           IF #rdrec.valid = TRUE THEN
               // store information of data record
               #readdata[0] := DINT_TO_BYTE(#RDREC_Function.INDEX); // ID of data record
               #readdata[1] := UINT_TO_BYTE(#rdrec.len);    // Length of data record
               #idpos := DINT#8;   // set start position within data
               MOVE_BLK(IN := #recorddata[0],
                        COUNT := #rdrec.len,
                        OUT => #readdata[#idpos]);
               #readlength := UINT_TO_INT(#rdrec.len);
               #sequencecontrol := 11;

           ELSIF #rdrec.error = TRUE THEN
               #ERROR := TRUE;
               #SF_STATUS := #rdrec.status;
               #sequencecontrol := 99; // function aborted with error
           ELSE
               ;
           END_IF; // store information of data record

       11:  // evaluate Consistency Check = Index 230d    
           #RDREC_Function(REQ := FALSE,
                           ID := #ID,
                           INDEX := DINT#230,
                           MLEN := UINT#0,
                           VALID => #rdrec.valid,
                           BUSY => #rdrec.busy,
                           ERROR => #rdrec.error,
                           STATUS => #rdrec.status,
                           LEN => #rdrec.len,
                           RECORD := #recorddata);

           IF #rdrec.valid = FALSE THEN
               #sequencecontrol := 12;
           ELSE
               ;
           END_IF;

       12:  // read Expected Port Configuration = Index 220d
           #STATUS := DW#16#00010220;
           #RDREC_Function(REQ := TRUE,
                           ID := #ID,
                           INDEX := DINT#220,
                           MLEN := UINT#0,
                           VALID => #rdrec.valid,
                           BUSY => #rdrec.busy,
                           ERROR => #rdrec.error,
                           STATUS => #rdrec.status,
                           LEN => #rdrec.len,
                           RECORD := #recorddata);

           IF #rdrec.valid = TRUE THEN
               // store information of data record
               #readdata[2] := DINT_TO_BYTE(#RDREC_Function.INDEX); // ID of data record
               #readdata[3] := UINT_TO_BYTE(#rdrec.len);    // Length of data record
               #idpos := #idpos + BYTE_TO_DINT(#readdata[1]);   // set start position within data
               MOVE_BLK(IN := #recorddata[0],
                        COUNT := #rdrec.len,
                        OUT => #readdata[#idpos]);
               #readlength := #readlength + UINT_TO_INT(#rdrec.len);
               #sequencecontrol := 13;

           ELSIF #rdrec.error = TRUE THEN
               #ERROR := TRUE;
               #SF_STATUS := #rdrec.status;
               #sequencecontrol := 99; // function aborted with error
           ELSE
               ;
           END_IF;

       13:  // evaluate Expected Port Configuration = Index 220d    
           #RDREC_Function(REQ := FALSE,
                           ID := #ID,
                           INDEX := DINT#220,
                           MLEN := UINT#0,
                           VALID => #rdrec.valid,
                           BUSY => #rdrec.busy,
                           ERROR => #rdrec.error,
                           STATUS => #rdrec.status,
                           LEN => #rdrec.len,
                           RECORD := #recorddata);
           IF #rdrec.valid = FALSE THEN
               #sequencecontrol := 14;
           END_IF;

       14:  // read IO Mapping = Index 222d
           #STATUS := DW#16#00010222;
           #RDREC_Function(REQ := TRUE,
                           ID := #ID,
                           INDEX := DINT#222,
                           MLEN := UINT#0,
                           VALID => #rdrec.valid,
                           BUSY => #rdrec.busy,
                           ERROR => #rdrec.error,
                           STATUS => #rdrec.status,
                           LEN => #rdrec.len,
                           RECORD := #recorddata);

           IF #rdrec.valid = TRUE THEN
               // store information of data record
               #readdata[4] := DINT_TO_BYTE(#RDREC_Function.INDEX); // ID of data record
               #readdata[5] := UINT_TO_BYTE(#rdrec.len);    // Length of data record
               #idpos := #idpos + BYTE_TO_DINT(#readdata[3]);   // set start position within data
               MOVE_BLK(IN := #recorddata[0],
                        COUNT := #rdrec.len,
                        OUT => #readdata[#idpos]);
               #readlength := #readlength + UINT_TO_INT(#rdrec.len);
               #sequencecontrol := 15;

           ELSIF #rdrec.error = TRUE THEN
               #ERROR := TRUE;
               #SF_STATUS := #rdrec.status;
               #sequencecontrol := 99; // function aborted with error
           ELSE
               ;
           END_IF;

       15:  // evaluate IO Mapping = Index 222d    
           #RDREC_Function(REQ := FALSE,
                           ID := #ID,
                           INDEX := DINT#222,
                           MLEN := UINT#0,
                           VALID => #rdrec.valid,
                           BUSY => #rdrec.busy,
                           ERROR => #rdrec.error,
                           STATUS => #rdrec.status,
                           LEN => #rdrec.len,
                           RECORD := #recorddata);
           IF #rdrec.valid = FALSE THEN
               #sequencecontrol := 16;
           END_IF;

       16:  // BACKUP complete and valid
           #RECORD_DATA := #readdata;
           #DONE_VALID := TRUE;
           #BUSY := FALSE;
           #ERROR := FALSE;
           #STATUS := DW#16#00010000;
           #SF_STATUS := DW#16#00000000;
           #RD_LEN := #readlength + INT#8;

           #sequencecontrol := 98;

   (*---------------------------------------------------------------------------------------------------------------------
               Write master parameter = RESTORE
   ---------------------------------------------------------------------------------------------------------------------*)
       20: // write Expected Port Configuration = Index 220d
           #STATUS := DW#16#00020220;
           #idpos := DINT#8 + BYTE_TO_DINT(#writedata[1]);  // position of data record 
           #wrrec.len := BYTE_TO_UINT(#writedata[3]);   // length of data record
           MOVE_BLK(IN := #writedata[#idpos],
                    COUNT := #wrrec.len,
                    OUT => #recorddata[0]);
           #WRREC_Function(REQ := TRUE,
                           ID := #ID,
                           INDEX := BYTE_TO_DINT(#writedata[2]),
                           LEN := #wrrec.len,
                           DONE => #wrrec.done,
                           BUSY => #wrrec.busy,
                           ERROR => #wrrec.error,
                           STATUS => #wrrec.status,
                           RECORD := #recorddata);
           // wait for finish writing Expected Port Configuration = Index 220d                
           IF #wrrec.done = TRUE THEN
               #sequencecontrol := 21;
           ELSIF #wrrec.error = TRUE THEN
               #ERROR := TRUE;
               #SF_STATUS := #wrrec.status;
               #sequencecontrol := 99; // function aborted with error
           ELSE
               ;
           END_IF;

       21:  // writing Expected Port Configuration finished    
           #WRREC_Function(REQ := FALSE,
                           ID := #ID,
                           INDEX := BYTE_TO_DINT(#writedata[2]),
                           LEN := #wrrec.len,
                           DONE => #wrrec.done,
                           BUSY => #wrrec.busy,
                           ERROR => #wrrec.error,
                           STATUS => #wrrec.status,
                           RECORD := #recorddata);
           IF #wrrec.done = FALSE THEN
               #sequencecontrol := 22;
           END_IF;

       22:  // write IO Mapping = Index 222d
           #STATUS := DW#16#00020222;
           #idpos := DINT#8 + BYTE_TO_DINT(#writedata[1]) + BYTE_TO_DINT(#writedata[3]);  // position of data record 
           #wrrec.len := BYTE_TO_UINT(#writedata[5]);   // length of data record
           MOVE_BLK(IN := #writedata[#idpos],
                    COUNT := #wrrec.len,
                    OUT => #recorddata[0]);
           #WRREC_Function(REQ := TRUE,
                           ID := #ID,
                           INDEX := BYTE_TO_DINT(#writedata[4]),
                           LEN := #wrrec.len,
                           DONE => #wrrec.done,
                           BUSY => #wrrec.busy,
                           ERROR => #wrrec.error,
                           STATUS => #wrrec.status,
                           RECORD := #recorddata);
           // wait for finish writing IO Mapping = Index 222d                
           IF #wrrec.done = TRUE THEN
               #sequencecontrol := 23;
           ELSIF #wrrec.error = TRUE THEN
               #ERROR := TRUE;
               #SF_STATUS := #wrrec.status;
               #sequencecontrol := 99;
           ELSE
               ;
           END_IF;

       23:  // writing IO Mapping finished    
           #WRREC_Function(REQ := FALSE,
                           ID := #ID,
                           INDEX := BYTE_TO_DINT(#writedata[4]),
                           LEN := #wrrec.len,
                           DONE => #wrrec.done,
                           BUSY => #wrrec.busy,
                           ERROR => #wrrec.error,
                           STATUS => #wrrec.status,
                           RECORD := #recorddata);
           IF #wrrec.done = FALSE THEN
               #sequencecontrol := 24;
           END_IF;

       24:  // write Consistency Check = Index 230d
           #STATUS := DW#16#00020230;
           #idpos := DINT#8;  // position of data record 
           #wrrec.len := BYTE_TO_UINT(#writedata[1]);   // length of data record
           MOVE_BLK(IN := #writedata[#idpos],
                    COUNT := #wrrec.len,
                    OUT => #recorddata[0]);
           #WRREC_Function(REQ := TRUE,
                           ID := #ID,
                           INDEX := BYTE_TO_DINT(#writedata[0]),
                           LEN := #wrrec.len,
                           DONE => #wrrec.done,
                           BUSY => #wrrec.busy,
                           ERROR => #wrrec.error,
                           STATUS => #wrrec.status,
                           RECORD := #recorddata);
           // wait for finish writing Consistency Check = Index 230d               
           IF #wrrec.done = TRUE THEN
               #sequencecontrol := 25;
           ELSIF #wrrec.error = TRUE THEN
               #ERROR := TRUE;
               #SF_STATUS := #wrrec.status;
               #sequencecontrol := 99;
           ELSE
               ;
           END_IF;

       25:  // writing ConsistencyCheck finished    
           #WRREC_Function(REQ := FALSE,
                           ID := #ID,
                           INDEX := BYTE_TO_DINT(#writedata[0]),
                           LEN := #wrrec.len,
                           DONE => #wrrec.done,
                           BUSY => #wrrec.busy,
                           ERROR => #wrrec.error,
                           STATUS => #wrrec.status,
                           RECORD := #recorddata);
           IF #wrrec.done = FALSE THEN
               #sequencecontrol := 26;
           END_IF;

       26:  // RESTORE complete and valid
           #DONE_VALID := TRUE;
           #BUSY := FALSE;
           #ERROR := FALSE;
           #STATUS := DW#16#00020000;
           #SF_STATUS := DW#16#00000000;
           #RD_LEN := INT#0;

           #sequencecontrol := 98;

   (*---------------------------------------------------------------------------------------------------------------------
               END of SEQUENCE CONTROL
   ---------------------------------------------------------------------------------------------------------------------*)
       98: // Function complete and finish without error
           #RDREC_Function(REQ := FALSE,
                           RECORD := #recorddata);
           #WRREC_Function(REQ := FALSE);
           IF #REQ = FALSE THEN
               #DONE_VALID := FALSE;
               #STATUS := DW#16#00000000;
               #SF_STATUS := DW#16#00000000;
               #RD_LEN := INT#0;
               #sequencecontrol := 0;
               #typeofrequest := 0;
           END_IF;

       99: // Function aborted with error
           #RDREC_Function(REQ := FALSE,
                           RECORD := #recorddata);
           #WRREC_Function(REQ := FALSE);
           #DONE_VALID := FALSE;
           #BUSY := FALSE;
           #RD_LEN := INT#0;
           #sequencecontrol := 0;
           #typeofrequest := 0;

       ELSE  // no relevant case, ready for new request
           ;
   END_CASE;
END_FUNCTION_BLOCK

FUNCTION_BLOCK "IO_LINK_DEVICE"   // FB50001, SCL
{ S7_Optimized_Access := 'TRUE' }
AUTHOR : SUP_FA
FAMILY : IO-Link
VERSION : 3.0
   VAR_INPUT
      REQ : Bool;   // Request Function / Neuer Auftrag
      ID : Hw_Io;   // Hardwarekennung des IOL-Master Moduls (HW_IO) aus HW-Konfiguration
      CAP : DInt := DINT#0;   // Client Access Point (CAP), bei ET200 immer 227 dez
      RD_WR : Bool;   // Lese und Schreibzugriff auf IO-Link Device 0: Lesen, 1: schreiben
      PORT : Int := INT#0;   // Port/ Kanalnummer an dem das IO-Link Device betrieben wird. (ET200 = 1 .. 4)
      IOL_INDEX : Int := INT#0;   // Adressparameter Index (IO-Link Device) 0..32767 IOL-D, 65535 port functions
      IOL_SUBINDEX : Int := INT#0;   // Adressparameter Subindex (IO-Link Device) 0 ges. Record; 1-255 einz. Parameter
      LEN : Int := INT#0;   // Länge der zu schreibenden Daten (Nettodaten)
   END_VAR
   VAR_OUTPUT
      DONE_VALID : Bool;   // Gültigkeit 0: Daten nicht gültig; 1: Daten gültig
      BUSY : Bool;   // 0: Auftrag abgeschlossen 1: Auftrag in Bearbeitung
      ERROR : Bool;   // Fehler Flag 0: kein Fehler; 1: Abbruch der Funktion mit Fehler
      STATUS : DWord := DW#16#00000000;   // DP/ PNIO - Fehlerstatus; ERROR Flag = 1 - detaillierter Kommunikationsfehlerstatus
      IOL_STATUS : DWord := DW#16#00000000;   // IO-Link Fehlerstatus; ERROR Flag = 1 - detaillierte IO-Link Fehlerstatus
      RD_LEN : Int := INT#0;   // Länge des gelesenen Datensatzes (Anzahl Bytes)
   END_VAR
   VAR_IN_OUT
      RECORD_IOL_DATA : Array[0..231] of Byte;   // Datenbereich für LESEN / SCHREIBEN (max. 232 Byte)
   END_VAR
   VAR
      RDREC_Function : RDREC;   // Funktion Datensatz lesen (ehemals SFB52)
      WRREC_Function : WRREC;   // Funktion Datensatz schreiben (ehemals SFB53)
      TP_poll : TP_TIME;   // Pollzeit für "Datensatz lesen"
      TON_monitoring : TON_TIME;   // Überwachungszeit für Aufträge
      rdrec : Struct   // interne Struktur für RDREC
         valid : Bool;
         busy : Bool;
         error : Bool;
         status : DWord;
         length : UInt;
      END_STRUCT;
      wrrec : Struct   // interne Struktur für WRREC
         length : UInt;
         done : Bool;
         busy : Bool;
         error : Bool;
         status : DWord;
      END_STRUCT;
      read : Struct   // Datenbereich für Lesedaten
         header : Struct
            CALL : Struct
               Extended_Function_Num : Byte := 16#8;
               Port : Byte;
               FI_Index : Word := 16#FE4A;
            END_STRUCT;
            IOL : Struct
               Control : Byte;
               Index_HighByte : Byte;
               Index_LowByte : Byte;
               Subindex : Byte;
            END_STRUCT;
         END_STRUCT;
         data : Array[0..231] of Byte;
      END_STRUCT;
      write : Struct   // Datenbereich für Schreibdaten
         header : Struct
            CALL : Struct
               Extended_Function_Num : Byte := 16#8;
               Port : Byte;
               FI_Index : Word := 16#FE4A;
            END_STRUCT;
            IOL : Struct
               Control : Byte;
               Index_HighByte : Byte;
               Index_LowByte : Byte;
               Subindex : Byte;
            END_STRUCT;
         END_STRUCT;
         data : Array[0..231] of Byte;
      END_STRUCT;
      sequencecontrol : Int := INT#0;
      typeofrequest : Int := INT#0;
      R_TRIG_REQ : Bool;   // Impuls für neuen Auftrag starten
      R_TRIG_REQ_old : Bool;   // Flankenmerker
      F_TRIG_poll : Bool;   // Impuls für Pollen "Datensatz lesen"
      F_TRIG_poll_old : Bool;   // Flankenmerker
   END_VAR
   VAR_TEMP
      retval : Int;   // Variable für Rückgabewerte von Funktionen
      tmpWORD : Word;   // Datentyp WORD zur temporären Verwendung
      tmpDWORD : DWord;   // Datentyp DWORD zur temporären Verwendung
      tmpINT : Int;   // Datentyp INT zur temporären Verwendung
      i : Int;   // Laufvariable für for-Schleifen
   END_VAR
BEGIN
   (*---------------------------------------------------------------------------------------------------------------------
   SIEMENS AG
   ©Copyright 2015. All Rights Reserved.
   -----------------------------------------------------------------------------------------------------------------------
   Limitation of liability
   This software was developed with largest care. However, the author can not guarantee, that the software runs under
   each version of STEP7 on each PLC flawlessly.
   There is no warranty for the software, to the extent permitted by applicable law. The copyright holder provides the
   software "as is" without warranty of any kind, either expressed or implied, including, but not limited to, the implied
   warranties of merchantability and fitness for a particular purpose. The entire risk as to the quality and performance
   of the software is with you. Should the software prove defective, you assume the cost of all necessary servicing,
   repair or correction. In no event unless required by applicable law will the copyright holder be liable to you for
   damages, including any general, special, incidental or consequential damages arising out of the use or inability to
   use the software (including but not limited to loss of data or data being rendered inaccurate or losses sustained by
   you or third parties or a failure of the software to operate with any other programs), even if such holder or other
   party has been advised of the possibility of such damages.
   Permission to use or copy this software for any purpose is hereby granted without fee, provided the above notices are
   retained on all copies. Permission to modify the code and to distribute modified code is granted, provided the above
   notices are retained, and a notice that the code was modified is included with the above copyright notice.
   -----------------------------------------------------------------------------------------------------------------------
   Functionality provided by this source (short description):
   Function block IO_LINK_DEVICE - used to read and write of acyclic data records on devices with IO-Link.
   Note:
   To read data records, the IO-Link master modules needs to know which data record is required. Therefore it is necessary
   to send at first a request via write data record (only header of 8 byte). As response the IO-Link master module
   will send the required data record.

   Status:     Released (tested)
   File name:  IO_LINK_DEVICE
   System :    SIMATIC S7-1200/1500
   Version :   3.0
   -----------------------------------------------------------------------------------------------------------------------
   Script to be stored on level ... in project (mark appropriate levels with [x] below)
   [ ] External
   [ ] All levels possible
   [x] Project level
   [ ] Controller level
   [ ] Device level
   [ ] Subobject level
   -----------------------------------------------------------------------------------------------------------------------
   Restrictions, known limitations:
   The limitation of 240 byte is based on PROFIBUS DP protocol. With PROFINET IO there wouldn't no limit but because of 
   compatibility reason it wasn't changed.
     - header =   8 byte
     - data   = 232 byte
   -----------------------------------------------------------------------------------------------------------------------
   Requirements, prerequisites, External resources used: nothing
   -----------------------------------------------------------------------------------------------------------------------
   Change log table (latest change is at the bottom OF the list):
   Version Date Changes applied
   V2.0.0 <2013-09-30> First created with TIA Portal V12 SP1
   V2.1.0 <2014-03-14> Upgrade system function 'WRREC' from V1.0 to V1.1 and released for TIA Portal V13
   V3.0.0 <2015-02-28> Upgrade and released for TIA Portal V13 SP1 (without backup/restore master parameter)
   ---------------------------------------------------------------------------------------------------------------------*)

   (*---------------------------------------------------------------------------------------------------------------------
   Description of programmed IO-Link error codes
   8000 = time out
   8001 = wrong port
   8002 = wrong index
   8003 = wrong subindex
   8005 = wrong length for write data record
   8006 = wrong length for read data record
   8052 = error during reading data record
   8053 = error during writing data record
   All other codes are coming from a higher level!
   ---------------------------------------------------------------------------------------------------------------------*)

   (*---------------------------------------------------------------------------------------------------------------------
               NEW REQUEST
   ---------------------------------------------------------------------------------------------------------------------*)
   // detection rising edge of "REQ"
   #R_TRIG_REQ := #REQ = TRUE AND #R_TRIG_REQ_old = FALSE;
   #R_TRIG_REQ_old := #REQ = TRUE;

   // start new request if not busy
   IF #R_TRIG_REQ = TRUE AND #sequencecontrol = 0 THEN
       // Freeze record ID and CAP
       #WRREC_Function.ID := #ID;
       #WRREC_Function.INDEX := #CAP;
       #RDREC_Function.ID := #ID;
       #RDREC_Function.INDEX := #CAP;

       // Initialize outputs
       #DONE_VALID := FALSE;
       #BUSY := TRUE;
       #ERROR := FALSE;
       #STATUS := DW#16#00000000;
       #IOL_STATUS := DW#16#00000000;
       #RD_LEN := INT#0;

       // Initialize data area
       #read.header.CALL.Port := B#16#0;
       #read.header.IOL.Index_LowByte := B#16#0;
       #read.header.IOL.Index_HighByte := B#16#0;
       #read.header.IOL.Subindex := B#16#0;
       #i := INT#0; // initialize loop counter      
       FOR #i := 0 TO 231 DO
           #write.data[#i] := B#16#0;
           #read.data[#i] := B#16#0;
       END_FOR;

   (*---------------------------------------------------------------------------------------------------------------------
       Setup IO-LINK Call needs a specific header
   ---------------------------------------------------------------------------------------------------------------------*)
   // setup CALL header
   #write.header.CALL.Extended_Function_Num := 16#08;  // extended function number (fix coded 08h)
   #write.header.CALL.Port := INT_TO_BYTE(#PORT);  // 1..63 = PORT number, 64..255=reserved
   #write.header.CALL.FI_Index := 65098;  // IOL-Header is following (fix coded 65098)

   // setup IOL header 
   // CONTROL = please see below at BODY
   // INDEX
   #write.header.IOL.Index_LowByte := INT_TO_BYTE(#IOL_INDEX);
   #tmpWORD := INT_TO_WORD(#IOL_INDEX);
   #tmpWORD := SHR(IN := #tmpWORD, N := 8);
   #write.header.IOL.Index_HighByte := WORD_TO_BYTE(#tmpWORD);
   // SUBINDEX
   #write.header.IOL.Subindex := INT_TO_BYTE(#IOL_SUBINDEX);

   // BODY (data max. 232 Byte, Array 0..231 of Byte) 
   IF #RD_WR = TRUE THEN
       // IO-Link write data record requested, copy data from "RECORD_IOL_DATA"
       #write.header.IOL.Control := B#16#02; // CONTROL B#16#02 = write data record
       #wrrec.length := INT_TO_UINT(#LEN) + UINT#8;  // data length header + data = IO-Link write data record
       #typeofrequest := 2; // write data record
       // copy IOL_RECORD_DATA in working area
       #i := INT#0;    // initialize loop counter 
       FOR #i := 0 TO #LEN - 1 DO
           #write.data[#i] := #RECORD_IOL_DATA[#i];
       END_FOR;
   ELSE
       // IO-Link read data record requested
       #write.header.IOL.Control := 16#03;  // CONTROL 16#03 = read data record
       #wrrec.length := UINT#8; // data length only header = IO-Link read data record
       #typeofrequest := 1; // read data record        
   END_IF;
   #sequencecontrol := 1;  // Start sequence
   ELSE
       ;
   END_IF;

   (*---------------------------------------------------------------------------------------------------------------------
               SEQUENCE CONTROL
   ---------------------------------------------------------------------------------------------------------------------*)
   CASE #sequencecontrol OF
       1:  // Check input parameter        
           IF #PORT < INT#1 OR #PORT > INT#63 THEN // PORT (Wrong port address = 0x8001)
               #ERROR := TRUE;
               #IOL_STATUS := DW#16#80010000;
               #sequencecontrol := 99; // aborting function with error
           ELSIF #IOL_INDEX < INT#1 OR #IOL_INDEX > INT#32767 THEN    // INDEX (Wrong index = 0x8002)
               #ERROR := TRUE;
               #IOL_STATUS := DW#16#80020000;
               #sequencecontrol := 99; // aborting function with error
           ELSIF #IOL_SUBINDEX < INT#0 OR #IOL_SUBINDEX > INT#255 THEN    // SUBINDEX (Wrong subindex = 0x8003)
               #ERROR := TRUE;
               #IOL_STATUS := DW#16#80030000;
               #sequencecontrol := 99; // aborting function with error
           ELSIF #typeofrequest = 2 AND (#LEN < 1 OR #LEN > 232) THEN  // LEN (wrong length for write data record = 0x8004)
               #ERROR := TRUE;
               #IOL_STATUS := DW#16#80050000;
               #sequencecontrol := 99; // aborting function with error
           ELSIF #typeofrequest = 1 AND (#LEN < 0 OR #LEN > 232) THEN  // LEN (wrong length for read data record = 0x8005)
               #ERROR := TRUE;
               #IOL_STATUS := DW#16#80060000;
               #sequencecontrol := 99; // aborting function with error
           ELSE    // all input parameter are right
               #sequencecontrol := 2;
           END_IF;

       2:  (*-------------------------------------------------------------------------------------------------------------
           WRREC = Write Data Record
           Note:
           To read data records, the IO-Link master modules needs to know which PORT is required. Therefore it is necessary
           to send at first a request via write data record (header, 8 byte). As response the IO-Link master module will 
           send the required data record.
           -------------------------------------------------------------------------------------------------------------*)
           #WRREC_Function(REQ := TRUE,
                           LEN := #wrrec.length,
                           DONE => #wrrec.done,
                           BUSY => #wrrec.busy,
                           ERROR => #wrrec.error,
                           STATUS => #wrrec.status,
                           RECORD := #write);
           // output status during write data record
           IF #wrrec.busy THEN
               #STATUS := #wrrec.status;
               #IOL_STATUS := DW#16#00020000;  // 0002 = writing in progress 
           ELSIF #wrrec.error THEN
               #tmpDWORD := #wrrec.status AND DW#16#00FFFF00;  // filter status
               IF #tmpDWORD = DW#16#0080C200 THEN    // if resource #BUSY (#STATUS=80C2), then ... 
                   #sequencecontrol := 3;  // ... repeat write data record
               ELSE
                   #ERROR := TRUE;
                   #STATUS := #wrrec.status;   // ... otherwise output error status of "WRREC"
                   #IOL_STATUS := DW#16#80530000;  // ... with note '8053' = error status of "WRREC"
                   #sequencecontrol := 99; // aborting function with error
               END_IF;
           ELSIF #wrrec.done = TRUE THEN   // wait for write data record finish without error
               #TP_poll(IN := TRUE,
                        PT := T#100ms);    // poll for response
               #sequencecontrol := 4;
           ELSE
               ;
           END_IF;

       3:  // repeat write data record because resource was busy
           #WRREC_Function(REQ := FALSE);
           #sequencecontrol := 2;

       4:  // wait and poll for response = Read Data Record (RDREC)
           #WRREC_Function(REQ := FALSE);
           #TP_poll(IN := TRUE,
                    PT := T#100ms);

           // if poll rate executed then start read data record (on falling edge)
           #F_TRIG_poll := #TP_poll.Q = FALSE AND #F_TRIG_poll_old = TRUE;
           #F_TRIG_poll_old := #TP_poll.Q = TRUE;

           // RDREC = Read Data Record
           #RDREC_Function(REQ := #F_TRIG_poll,
                           MLEN := UINT#0, // length = 0 = read all data which are available
                           VALID => #rdrec.valid,
                           BUSY => #rdrec.busy,
                           ERROR => #rdrec.error,
                           STATUS => #rdrec.status,
                           LEN => #rdrec.length,
                           RECORD := #read);
           // output status during read data record
           IF #rdrec.busy THEN
               #STATUS := #rdrec.status;
               #IOL_STATUS := DW#16#00030000; // 16#0003 = reading in progress
           ELSIF #rdrec.error = TRUE THEN
               #tmpDWORD := #rdrec.status AND DW#16#00FFFF00;  // filter status
               IF #tmpDWORD = DW#16#0080C200 THEN  // if resource busy (status=80C2), then ... 
                   #sequencecontrol := 5;  // ... repeat read data record / continue polling
               ELSE
                   #ERROR := TRUE;
                   #STATUS := #rdrec.status;   // ... otherwise output error code of "RDREC"
                   #IOL_STATUS := DW#16#80520000;  // ... with note '8052' = error status of "RDREC"
                   #sequencecontrol := 99; // aborting function with error
               END_IF;
           ELSIF #rdrec.valid THEN
               IF  // check the response wether it matches the request (compare PORT, INDEX and SUBINDEX)
                   (#write.header.CALL.Port <> #read.header.CALL.Port) OR
                   (#write.header.IOL.Index_HighByte <> #read.header.IOL.Index_HighByte) OR
                   (#write.header.IOL.Index_LowByte <> #read.header.IOL.Index_LowByte) OR
                   (#write.header.IOL.Subindex <> #read.header.IOL.Subindex)
               THEN    // read data record don't match the request
                   #ERROR := TRUE;
                   #STATUS := #rdrec.status;
                   #IOL_STATUS := DW#16#70000000;  // output status '7000', no consistent data
                   #sequencecontrol := 99; // aborting function with error
               ELSIF #read.header.IOL.Control = B#16#80 THEN   // check the response for IO-Link errors
                   // State 0x80 = IOL_CALL_RES PDU shows IO-Link error detect
                   #ERROR := TRUE;
                   #STATUS := DW#16#00000000;
                   #IOL_STATUS.%B3 := #read.data[0];   // IO-Link master error code
                   #IOL_STATUS.%B2 := #read.data[1];   // IO-Link master error code
                   #IOL_STATUS.%B1 := #read.data[2];  // IO-Link device error code
                   #IOL_STATUS.%B0 := #read.data[3];  // IO-Link device additional error code

                   #sequencecontrol := 99; // aborting function with error
               ELSE    // read data are valid = output
                   #DONE_VALID := TRUE;
                   #BUSY := FALSE;
                   #ERROR := FALSE;
                   #STATUS := DW#16#00000000;
                   #IOL_STATUS := DW#16#00000000;  // request finished

                   IF #typeofrequest = 1 THEN
                       #RD_LEN := UINT_TO_INT(#rdrec.length - UINT#8);  // device parameter cover header and data,
                       // only data will be output
                       #i := INT#0; // initialize loop counter
                       FOR #i := 0 TO UINT_TO_INT(#rdrec.length - UINT#8 - UINT#1) DO
                           #RECORD_IOL_DATA[#i] := #read.data[#i];
                       END_FOR;
                   ELSE
                       ;
                   END_IF;
                   #sequencecontrol := 98;
               END_IF;
           ELSE
               ;
           END_IF;

       5:  // poll again for response because resource was busy
           #TP_poll(IN := FALSE,
                    PT := T#100ms);
           #RDREC_Function(REQ := FALSE,
                           RECORD := #read);
           #sequencecontrol := 4;  // ... repeat read data record / continue polling   

       98: // request done successfully
           #TP_poll(IN := FALSE,
                    PT := T#100ms);
           #RDREC_Function(REQ := FALSE,
                           RECORD := #read);
           IF #REQ = FALSE THEN
               #DONE_VALID := FALSE;
               #BUSY := FALSE;
               #ERROR := FALSE;
               #RD_LEN := INT#0;
               #STATUS := DW#16#00000000;
               #IOL_STATUS := DW#16#00010000; // ready for new request
               #sequencecontrol := 0;
               #typeofrequest := 0;
           ELSE
               ;
           END_IF;

       99: // Function aborted with error
           #TP_poll(IN := FALSE,
                    PT := T#100ms);
           #WRREC_Function(REQ := FALSE);
           #RDREC_Function(REQ := FALSE,
                           RECORD := #read);
           #DONE_VALID := FALSE;
           #BUSY := FALSE;
           #RD_LEN := INT#0;
           #sequencecontrol := 0;
           #typeofrequest := 0;

       ELSE  // no relevant case, ready for new request
           #WRREC_Function(REQ := FALSE);
           #RDREC_Function(REQ := FALSE,
                           RECORD := #read);
           #TP_poll(IN := FALSE,
                    PT := T#100ms);
           #TON_monitoring(IN := FALSE,
                           PT := T#20s);
           #sequencecontrol := 0;
           #typeofrequest := 0;
   END_CASE;

   (*---------------------------------------------------------------------------------------------------------------------
               MONITORING
   ---------------------------------------------------------------------------------------------------------------------*)
   #TON_monitoring(IN := #sequencecontrol > 0 AND #sequencecontrol < 98,
                   PT := T#20s);
   IF #TON_monitoring.Q THEN
       #ERROR := TRUE;
       #IOL_STATUS := DW#16#80000000; // request time out       
       #sequencecontrol := 99; // aborting function with error
   END_IF;
END_FUNCTION_BLOCK

FUNCTION "SetzePufferstand" : Void   // FC1, SCL
{ S7_Optimized_Access := 'TRUE' }
VERSION : 0.1
   VAR_INPUT
      SmLiNr : Int;
      Pufferstand : Int;
   END_VAR
   VAR_TEMP
      PufferSetzwert : Int;
      SmartlightNumber : Int;
      Temp_1 : Array[0..1] of Byte;
   END_VAR
   VAR CONSTANT
      Adresse : Word;
   END_VAR
BEGIN
   #SmartlightNumber := #SmLiNr - 1;
   "DB_Station4_Puffer".Pufferstand[#SmartlightNumber] := #Pufferstand;
   IF TRUE THEN //TODO Wertebereich pruefen
       //Pruefen der eingestellten Granularitaet vor dem Setzen.
       //Neuberechung, wenn ungueltig
       IF "DB_Station4_Puffer".Faktoren[#SmartlightNumber] <= 0 THEN
           "BestimmeGranularitaet"(#SmLiNr);
       END_IF;
       //Berechnen des gesetzten Bytes am Smartlight
       #PufferSetzwert := #Pufferstand*"DB_Station4_Puffer".Faktoren[#SmartlightNumber];
       //Setzen des Bytes am Smartlight
       CASE #SmLiNr OF
           1:  // Smartlight 1 (klein)
               "OutByteM1P2.1" := INT_TO_BYTE(#PufferSetzwert);
           2:  // Smartlight 2 (gross)
               "OutByteM1P3_Level8bit" := INT_TO_BYTE(#PufferSetzwert);
       END_CASE;
   END_IF;
END_FUNCTION

FUNCTION "BestimmeGranularitaet" : Void   // FC2, SCL
{ S7_Optimized_Access := 'TRUE' }
VERSION : 0.1
   VAR_INPUT
      SmLiNr : Int;
   END_VAR
   VAR_TEMP
      SmartlightNumber : Int;
      MaxPuffer : Int;
   END_VAR
BEGIN
   #SmartlightNumber := #SmLiNr-1;
   IF "DB_Station4_Puffer".CONST_MAXPUFFER[#SmartlightNumber] <= 0 THEN
       #MaxPuffer := "DB_Konstanten".DEFAULT_STATION4_MAXPUFFER[#SmartlightNumber];
   ELSE
       #MaxPuffer := "DB_Station4_Puffer".CONST_MAXPUFFER[#SmartlightNumber];
   END_IF;
   "DB_Station4_Puffer".Faktoren[#SmartlightNumber] := FLOOR(256 / #MaxPuffer);
END_FUNCTION

FUNCTION "Lese8Byte" : Void   // FC3, SCL
{ S7_Optimized_Access := 'TRUE' }
VERSION : 0.1
   VAR_INPUT
      Adresse : Hw_Io;
   END_VAR
   VAR_OUTPUT
      Wert : Array[0..7] of Byte;
   END_VAR
   VAR_TEMP
      i : Int;
      index : Int;
      BeginnAdresse : Int;
      EndeAdresse : Int;
      temp : Int;
   END_VAR
BEGIN
   #i := 0;
   #temp := RD_ADDR(LADDR:=#Adresse,PIADDR => #BeginnAdresse,PICount => #temp,PQADDR => #temp,PQCount=> #temp);
   #BeginnAdresse := #BeginnAdresse + 1;
   #EndeAdresse := #BeginnAdresse + 7;
   FOR #index := #BeginnAdresse TO #EndeAdresse DO
       #Wert[#i] := PEEK(area := 16#81, dbNumber := 0, byteOffset := #index);
       #i := #i + 1;
   END_FOR;
END_FUNCTION

FUNCTION "LeseID" : Void   // FC4, SCL
{ S7_Optimized_Access := 'TRUE' }
VERSION : 0.1
   VAR_INPUT
      Adresse : Hw_Io;
   END_VAR
   VAR_OUTPUT
      ID : String;
   END_VAR
   VAR_TEMP
      temp : Int;
      BeginnAdresse : Int;
      EndeAdresse : Int;
      index : Int;
      s : String;
      s2 : String;
   END_VAR
BEGIN
   #ID := '';
   #temp := RD_ADDR(LADDR := #Adresse, PIADDR => #BeginnAdresse, PICount => #temp, PQADDR => #temp, PQCount => #temp);
   #BeginnAdresse := #BeginnAdresse + 1;
   #EndeAdresse := #BeginnAdresse + 7;
   FOR #index := #BeginnAdresse TO #EndeAdresse DO
       #s := S_CONV(BYTE_TO_INT(PEEK(area := 16#81, dbNumber := 0, byteOffset := #index)));
       #s := RIGHT(IN := #s, L := LEN(IN := #s)-1);
       #ID := CONCAT(IN1 := #ID,IN2 := #s);
   END_FOR;
END_FUNCTION

ORGANIZATION_BLOCK "Main"   // OB1, LAD, ProgramCycle
TITLE = "Main Program Sweep (Cycle)"
{ S7_Optimized_Access := 'TRUE' }
VERSION : 0.1
   VAR_INPUT
      Initial_Call : Bool;   // Initial call of this OB
      Remanence : Bool;   // =True, if remanent data are available
   END_VAR
   VAR_TEMP
      i : Int;
      Adresse : Hw_Any;
      KennungVorhanden : UInt;
      KennungFehler : UInt;
      ZustandVorhanden : Bool;
      ZustandFehler : Bool;
      temp : Int;
      KennungDeaktivieren : USInt;
      tempbool : Array[0..19] of Bool;
      KennungAbfrage : USInt;
      tempBoolAct : Bool;
      testbool : Bool;
   END_VAR
   VAR_TEMP   // added for the SCL form of the ladder/FBD networks
      _w1 : Bool;
      _w2 : Bool;
      _w3 : Bool;
      _w4 : Bool;
      _w5 : Bool;
      _w6 : Bool;
      _w7 : Bool;
      _w8 : Bool;
      _w9 : Bool;
      _w10 : Bool;
      _w11 : Bool;
      _w12 : Bool;
      _w13 : Bool;
      _w14 : Bool;
      _w15 : Bool;
   END_VAR
BEGIN

REGION Network 1: Station2/Port1
   // Setzen der Werte für den entsprechenden Datenbaustein
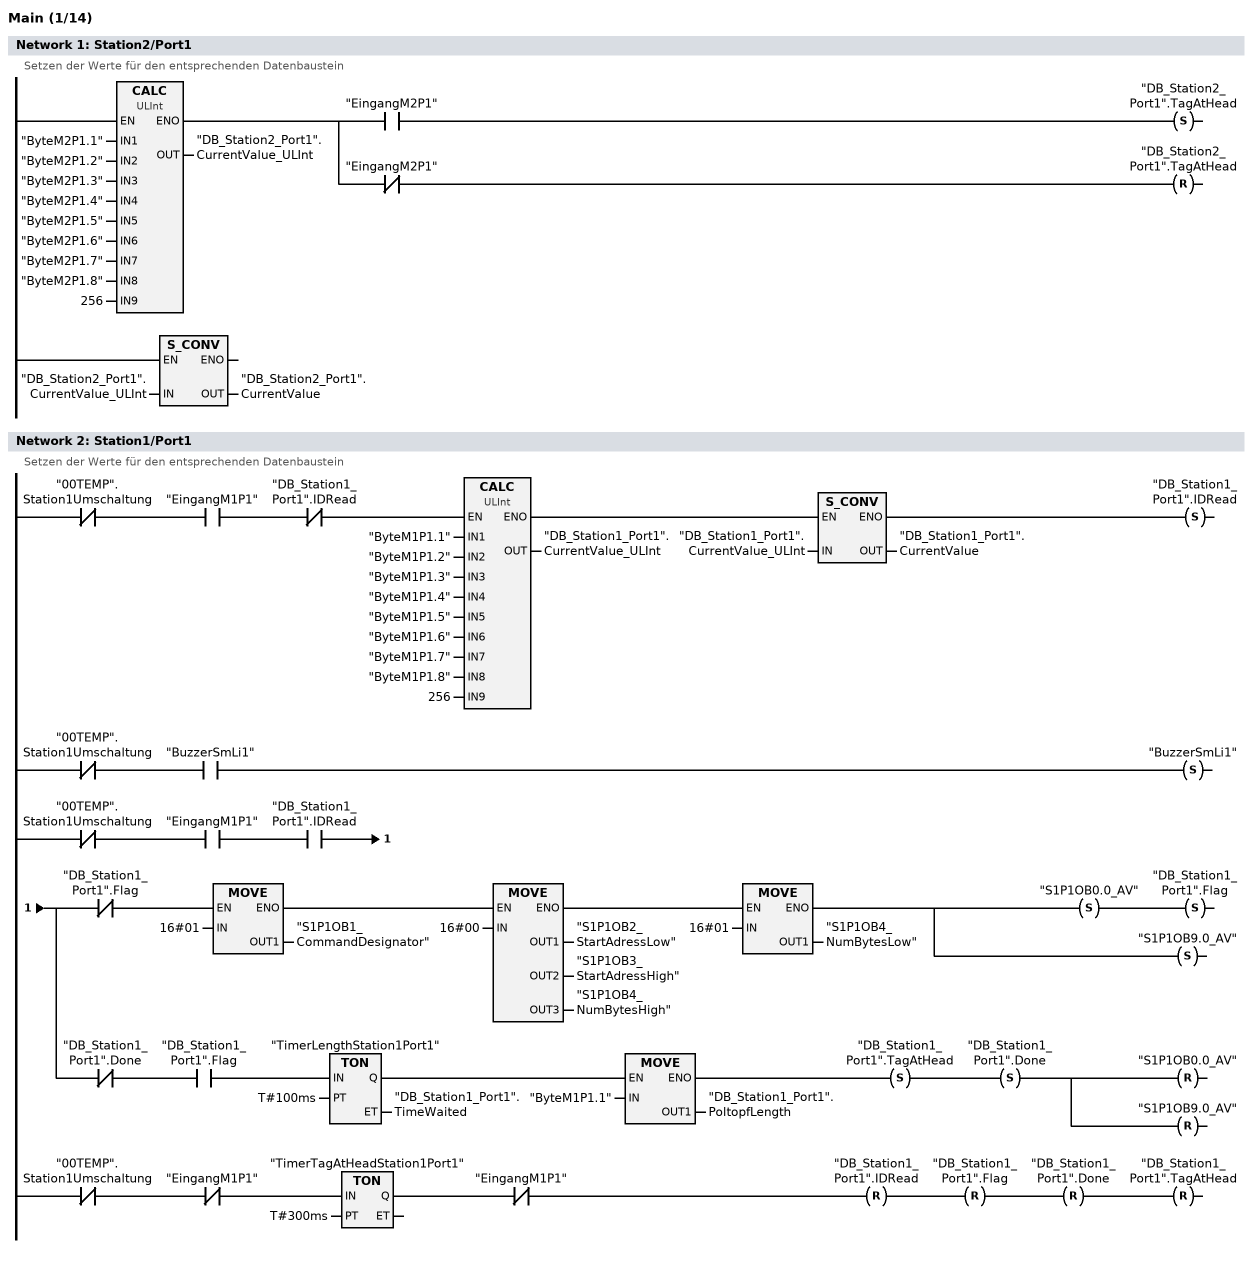
   CALC(in1 := "ByteM2P1.1",
        in2 := "ByteM2P1.2",
        in3 := "ByteM2P1.3",
        in4 := "ByteM2P1.4",
        in5 := "ByteM2P1.5",
        in6 := "ByteM2P1.6",
        in7 := "ByteM2P1.7",
        in8 := "ByteM2P1.8",
        in9 := 256,
        out => "DB_Station2_Port1".CurrentValue_ULInt);
   IF "EingangM2P1" THEN "DB_Station2_Port1".TagAtHead := TRUE; END_IF;
   IF NOT "EingangM2P1" THEN "DB_Station2_Port1".TagAtHead := FALSE; END_IF;
   "DB_Station2_Port1".CurrentValue := S_CONV(IN := "DB_Station2_Port1".CurrentValue_ULInt);
END_REGION

REGION Network 2: Station1/Port1
   // Setzen der Werte für den entsprechenden Datenbaustein
   #_w1 := NOT "00TEMP".Station1Umschaltung AND "EingangM1P1" AND NOT "DB_Station1_Port1".IDRead;
   IF #_w1 THEN
       CALC(in1 := "ByteM1P1.1",
            in2 := "ByteM1P1.2",
            in3 := "ByteM1P1.3",
            in4 := "ByteM1P1.4",
            in5 := "ByteM1P1.5",
            in6 := "ByteM1P1.6",
            in7 := "ByteM1P1.7",
            in8 := "ByteM1P1.8",
            in9 := 256,
            out => "DB_Station1_Port1".CurrentValue_ULInt);
       "DB_Station1_Port1".CurrentValue := S_CONV(IN := "DB_Station1_Port1".CurrentValue_ULInt);
       "DB_Station1_Port1".IDRead := TRUE;
   END_IF;
   IF NOT "00TEMP".Station1Umschaltung AND "BuzzerSmLi1" THEN "BuzzerSmLi1" := TRUE; END_IF;
   #_w2 := NOT "00TEMP".Station1Umschaltung AND "EingangM1P1" AND "DB_Station1_Port1".IDRead;
   IF #_w2 AND NOT "DB_Station1_Port1".Flag THEN
       "S1P1OB1_CommandDesignator" := 16#01;
       "S1P1OB2_StartAdressLow" := 16#00;
       "S1P1OB3_StartAdressHigh" := 16#00;
       "S1P1OB4_NumBytesHigh" := 16#00;
       "S1P1OB4_NumBytesLow" := 16#01;
       "S1P1OB0.0_AV" := TRUE;
   END_IF;
   #_w3 := #_w2 AND NOT "DB_Station1_Port1".Flag;
   IF #_w3 THEN
       "DB_Station1_Port1".Flag := TRUE;
       "S1P1OB9.0_AV" := TRUE;
   END_IF;
   "TimerLengthStation1Port1".TON(IN := #_w2 AND NOT "DB_Station1_Port1".Done AND "DB_Station1_Port1".Flag,
                           PT := T#100ms,
                           ET => "DB_Station1_Port1".TimeWaited);
   IF "TimerLengthStation1Port1".Q THEN
       "DB_Station1_Port1".PoltopfLength := "ByteM1P1.1";
       "DB_Station1_Port1".TagAtHead := TRUE;
       "DB_Station1_Port1".Done := TRUE;
       "S1P1OB0.0_AV" := FALSE;
       "S1P1OB9.0_AV" := FALSE;
   END_IF;
   "TimerTagAtHeadStation1Port1".TON(IN := NOT "00TEMP".Station1Umschaltung AND NOT "EingangM1P1",
                           PT := T#300ms);
   IF "TimerTagAtHeadStation1Port1".Q AND NOT "EingangM1P1" THEN
       "DB_Station1_Port1".IDRead := FALSE;
       "DB_Station1_Port1".Flag := FALSE;
       "DB_Station1_Port1".Done := FALSE;
       "DB_Station1_Port1".TagAtHead := FALSE;
   END_IF;
END_REGION

REGION Network 3: Station 1 Port 1 Temp
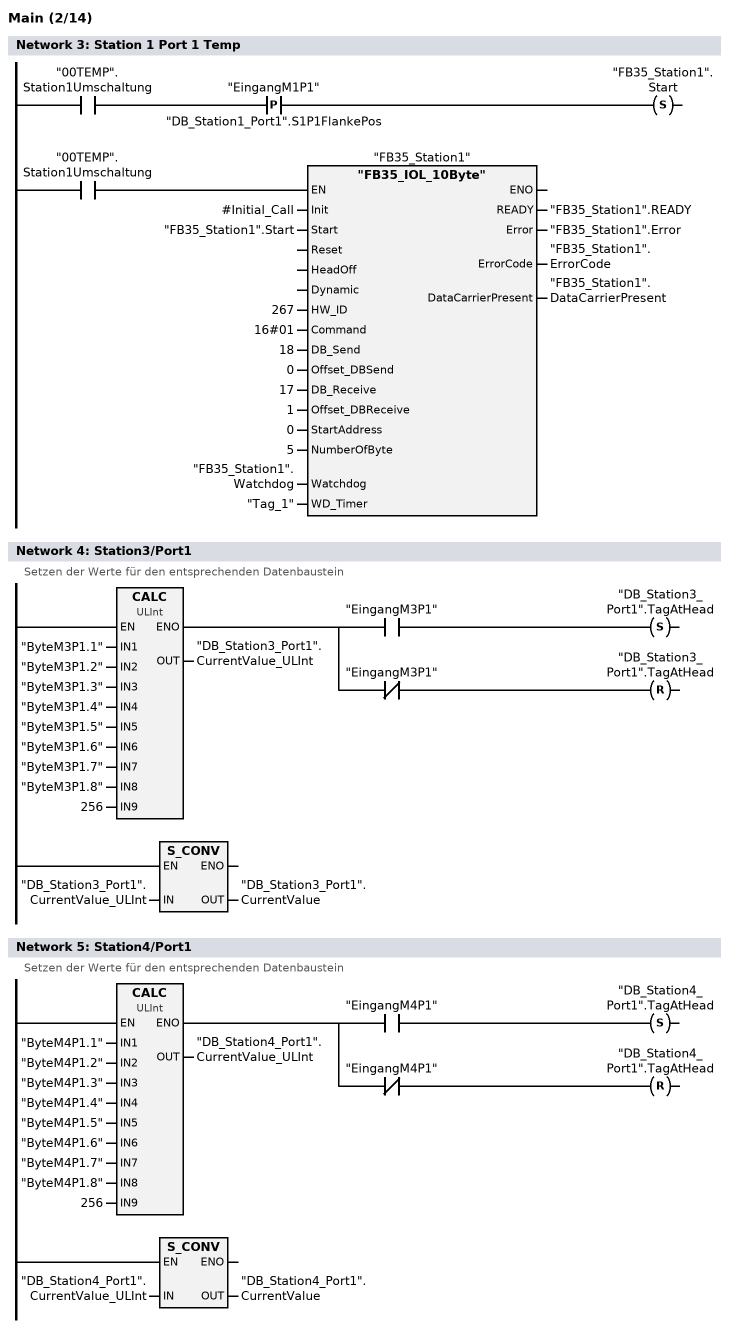
   RUNG wire#powerrail
      Contact( "00TEMP".Station1Umschaltung )
      P_Contact(operand := "EingangM1P1", bit := "DB_Station1_Port1".S1P1FlankePos)
      S_Coil( "FB35_Station1".Start )
   END_RUNG
   RUNG wire#powerrail
      Contact( "00TEMP".Station1Umschaltung )
      "FB35_Station1"(Init := #Initial_Call, Start := "FB35_Station1".Start, Reset :=, HeadOff :=, Dynamic :=, HW_ID := 267, Command := 16#01, DB_Send := 18, Offset_DBSend := 0, DB_Receive := 17, Offset_DBReceive := 1, StartAddress := 0, NumberOfByte := 5, Watchdog := "FB35_Station1".Watchdog, WD_Timer := "Tag_1", READY => "FB35_Station1".READY, Error => "FB35_Station1".Error, ErrorCode => "FB35_Station1".ErrorCode, DataCarrierPresent => "FB35_Station1".DataCarrierPresent)
   END_RUNG
   // the same network as SCL:
   #_w1 := "00TEMP".Station1Umschaltung AND "EingangM1P1" AND NOT "DB_Station1_Port1".S1P1FlankePos;   // rising edge of "EingangM1P1"
   "DB_Station1_Port1".S1P1FlankePos := "EingangM1P1";
   IF #_w1 THEN "FB35_Station1".Start := TRUE; END_IF;
   IF "00TEMP".Station1Umschaltung THEN
       "FB35_Station1"(Init := #Initial_Call,   // "FB35_IOL_10Byte"
                       Start := "FB35_Station1".Start,
                       HW_ID := 267,
                       Command := 16#01,
                       DB_Send := 18,
                       Offset_DBSend := 0,
                       DB_Receive := 17,
                       Offset_DBReceive := 1,
                       StartAddress := 0,
                       NumberOfByte := 5,
                       Watchdog := "FB35_Station1".Watchdog,
                       WD_Timer := "Tag_1",
                       READY => "FB35_Station1".READY,
                       Error => "FB35_Station1".Error,
                       ErrorCode => "FB35_Station1".ErrorCode,
                       DataCarrierPresent => "FB35_Station1".DataCarrierPresent);
   END_IF;
END_REGION

REGION Network 4: Station3/Port1
   // Setzen der Werte für den entsprechenden Datenbaustein
   CALC(in1 := "ByteM3P1.1",
        in2 := "ByteM3P1.2",
        in3 := "ByteM3P1.3",
        in4 := "ByteM3P1.4",
        in5 := "ByteM3P1.5",
        in6 := "ByteM3P1.6",
        in7 := "ByteM3P1.7",
        in8 := "ByteM3P1.8",
        in9 := 256,
        out => "DB_Station3_Port1".CurrentValue_ULInt);
   IF "EingangM3P1" THEN "DB_Station3_Port1".TagAtHead := TRUE; END_IF;
   IF NOT "EingangM3P1" THEN "DB_Station3_Port1".TagAtHead := FALSE; END_IF;
   "DB_Station3_Port1".CurrentValue := S_CONV(IN := "DB_Station3_Port1".CurrentValue_ULInt);
END_REGION

REGION Network 5: Station4/Port1
   // Setzen der Werte für den entsprechenden Datenbaustein
   CALC(in1 := "ByteM4P1.1",
        in2 := "ByteM4P1.2",
        in3 := "ByteM4P1.3",
        in4 := "ByteM4P1.4",
        in5 := "ByteM4P1.5",
        in6 := "ByteM4P1.6",
        in7 := "ByteM4P1.7",
        in8 := "ByteM4P1.8",
        in9 := 256,
        out => "DB_Station4_Port1".CurrentValue_ULInt);
   IF "EingangM4P1" THEN "DB_Station4_Port1".TagAtHead := TRUE; END_IF;
   IF NOT "EingangM4P1" THEN "DB_Station4_Port1".TagAtHead := FALSE; END_IF;
   "DB_Station4_Port1".CurrentValue := S_CONV(IN := "DB_Station4_Port1".CurrentValue_ULInt);
END_REGION

REGION Network 6: Station4/Port1 lesen und entsprechendes SmartLight an Station1 und 11 hochzaehlen
   // Abfrage ob langer oder kurzer Poltopf - beide Smartlights an Station1 oder 11
   // Der Schreblesekopf muss entsprechend auf "send data starting at startadress" gesetzt sein!
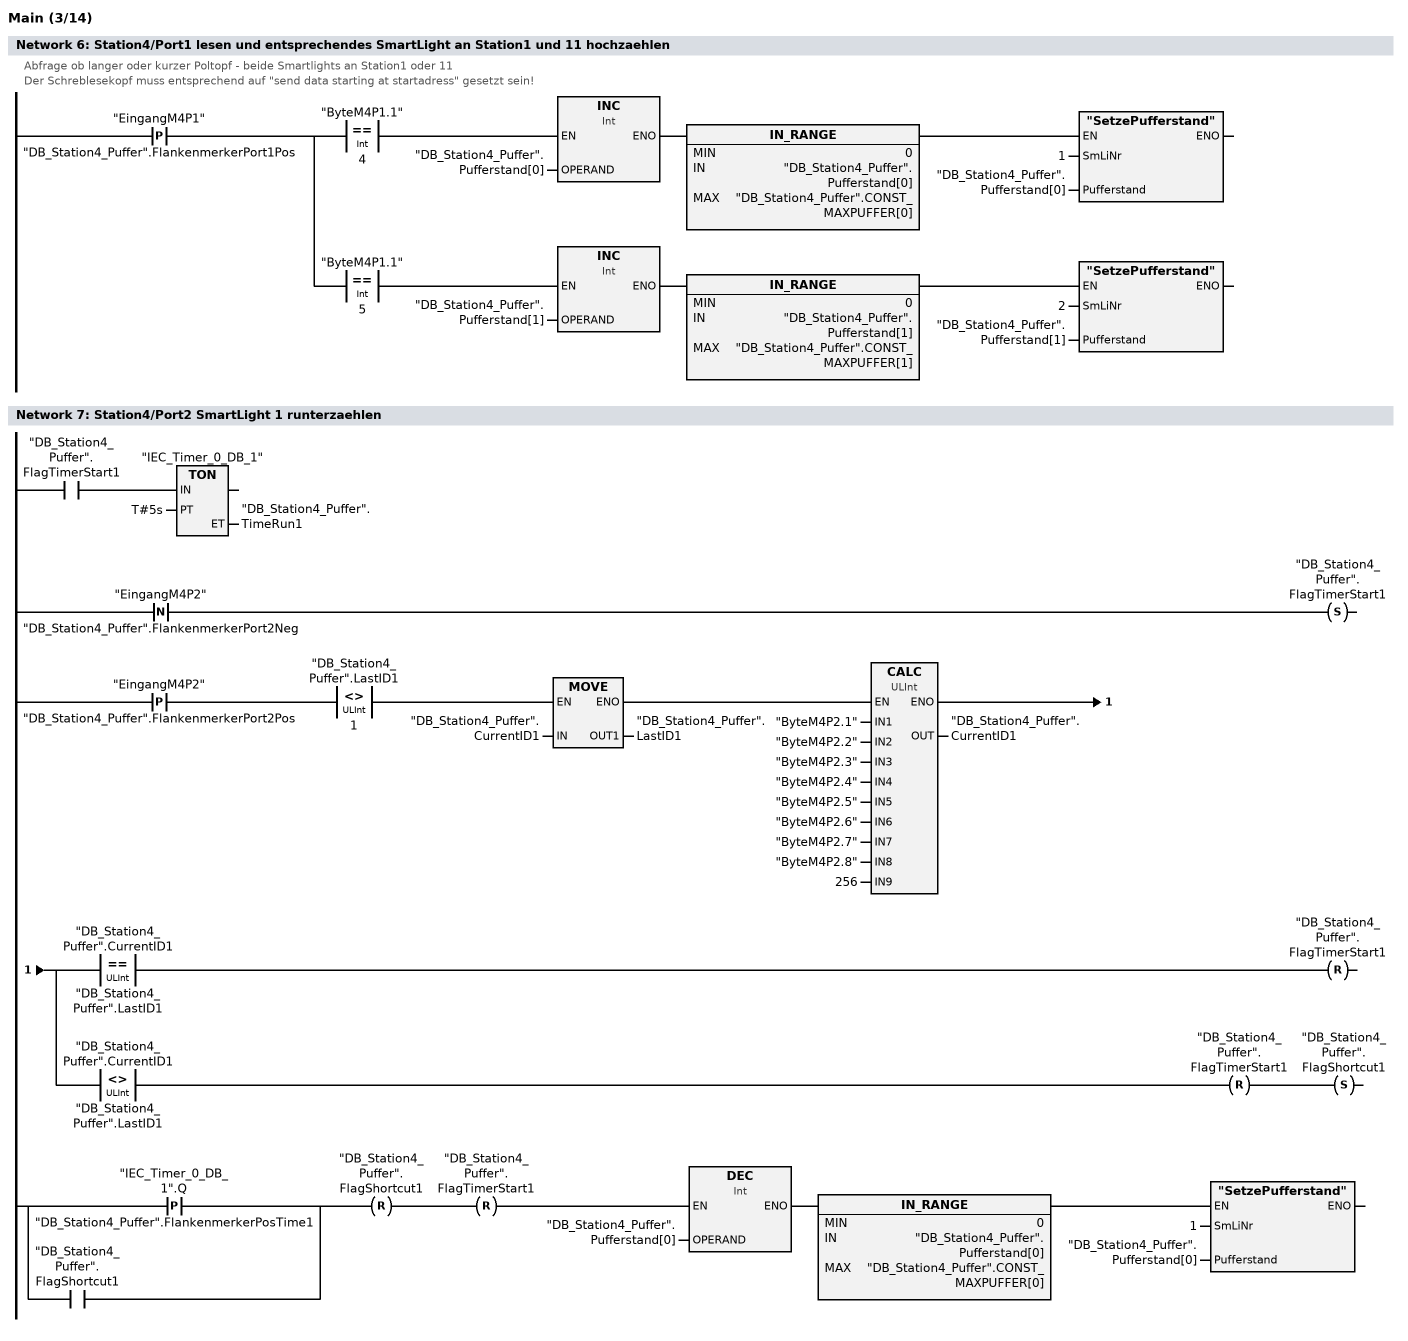
   RUNG wire#powerrail
      P_Contact(operand := "EingangM4P1", bit := "DB_Station4_Puffer".FlankenmerkerPort1Pos)
      wire#w1
      { S7_Templates := "SrcType := Int" } EQ_Contact(in1 := "ByteM4P1.1", in2 := 4)
      { S7_Templates := "DestType := Int" } Inc( "DB_Station4_Puffer".Pufferstand[0] )
      { S7_Templates := "SrcType := Int" } InRange(min := 0, in := "DB_Station4_Puffer".Pufferstand[0], max := "DB_Station4_Puffer".CONST_MAXPUFFER[0])
      "SetzePufferstand"(SmLiNr := 1, Pufferstand := "DB_Station4_Puffer".Pufferstand[0])
   END_RUNG
   RUNG wire#w1
      { S7_Templates := "SrcType := Int" } EQ_Contact(in1 := "ByteM4P1.1", in2 := 5)
      { S7_Templates := "DestType := Int" } Inc( "DB_Station4_Puffer".Pufferstand[1] )
      { S7_Templates := "SrcType := Int" } InRange(min := 0, in := "DB_Station4_Puffer".Pufferstand[1], max := "DB_Station4_Puffer".CONST_MAXPUFFER[1])
      "SetzePufferstand"(SmLiNr := 2, Pufferstand := "DB_Station4_Puffer".Pufferstand[1])
   END_RUNG
   // the same network as SCL:
   #_w1 := "EingangM4P1" AND NOT "DB_Station4_Puffer".FlankenmerkerPort1Pos;   // rising edge of "EingangM4P1"
   "DB_Station4_Puffer".FlankenmerkerPort1Pos := "EingangM4P1";
   #_w2 := #_w1 AND ("ByteM4P1.1" = 4);
   IF #_w2 THEN "DB_Station4_Puffer".Pufferstand[0] := "DB_Station4_Puffer".Pufferstand[0] + 1; END_IF;
   IF #_w2 AND (0 <= "DB_Station4_Puffer".Pufferstand[0]) AND ("DB_Station4_Puffer".Pufferstand[0] <= "DB_Station4_Puffer".CONST_MAXPUFFER[0]) THEN
       "SetzePufferstand"(SmLiNr := 1, Pufferstand := "DB_Station4_Puffer".Pufferstand[0]);
   END_IF;
   #_w3 := #_w1 AND ("ByteM4P1.1" = 5);
   IF #_w3 THEN "DB_Station4_Puffer".Pufferstand[1] := "DB_Station4_Puffer".Pufferstand[1] + 1; END_IF;
   IF #_w3 AND (0 <= "DB_Station4_Puffer".Pufferstand[1]) AND ("DB_Station4_Puffer".Pufferstand[1] <= "DB_Station4_Puffer".CONST_MAXPUFFER[1]) THEN
       "SetzePufferstand"(SmLiNr := 2, Pufferstand := "DB_Station4_Puffer".Pufferstand[1]);
   END_IF;
END_REGION

REGION Network 7: Station4/Port2 SmartLight 1 runterzaehlen
   "IEC_Timer_0_DB_1".TON(IN := "DB_Station4_Puffer".FlagTimerStart1,
                          PT := T#5s,
                          ET => "DB_Station4_Puffer".TimeRun1);
   #_w1 := NOT "EingangM4P2" AND "DB_Station4_Puffer".FlankenmerkerPort2Neg;   // falling edge of "EingangM4P2"
   "DB_Station4_Puffer".FlankenmerkerPort2Neg := "EingangM4P2";
   IF #_w1 THEN "DB_Station4_Puffer".FlagTimerStart1 := TRUE; END_IF;
   #_w2 := "EingangM4P2" AND NOT "DB_Station4_Puffer".FlankenmerkerPort2Pos;   // rising edge of "EingangM4P2"
   "DB_Station4_Puffer".FlankenmerkerPort2Pos := "EingangM4P2";
   #_w3 := #_w2 AND ("DB_Station4_Puffer".LastID1 <> 1);
   IF #_w3 THEN
       "DB_Station4_Puffer".LastID1 := "DB_Station4_Puffer".CurrentID1;
       CALC(in1 := "ByteM4P2.1",
            in2 := "ByteM4P2.2",
            in3 := "ByteM4P2.3",
            in4 := "ByteM4P2.4",
            in5 := "ByteM4P2.5",
            in6 := "ByteM4P2.6",
            in7 := "ByteM4P2.7",
            in8 := "ByteM4P2.8",
            in9 := 256,
            out => "DB_Station4_Puffer".CurrentID1);
   END_IF;
   IF #_w3 AND ("DB_Station4_Puffer".CurrentID1 = "DB_Station4_Puffer".LastID1) THEN
       "DB_Station4_Puffer".FlagTimerStart1 := FALSE;
   END_IF;
   IF #_w3 AND ("DB_Station4_Puffer".CurrentID1 <> "DB_Station4_Puffer".LastID1) THEN
       "DB_Station4_Puffer".FlagTimerStart1 := FALSE;
       "DB_Station4_Puffer".FlagShortcut1 := TRUE;
   END_IF;
   #_w4 := "IEC_Timer_0_DB_1".Q AND NOT "DB_Station4_Puffer".FlankenmerkerPosTime1;   // rising edge of "IEC_Timer_0_DB_1".Q
   "DB_Station4_Puffer".FlankenmerkerPosTime1 := "IEC_Timer_0_DB_1".Q;
   #_w5 := #_w4 OR "DB_Station4_Puffer".FlagShortcut1;
   IF #_w5 THEN
       "DB_Station4_Puffer".FlagShortcut1 := FALSE;
       "DB_Station4_Puffer".FlagTimerStart1 := FALSE;
       "DB_Station4_Puffer".Pufferstand[0] := "DB_Station4_Puffer".Pufferstand[0] - 1;
   END_IF;
   IF #_w5 AND (0 <= "DB_Station4_Puffer".Pufferstand[0]) AND ("DB_Station4_Puffer".Pufferstand[0] <= "DB_Station4_Puffer".CONST_MAXPUFFER[0]) THEN
       "SetzePufferstand"(SmLiNr := 1, Pufferstand := "DB_Station4_Puffer".Pufferstand[0]);
   END_IF;
END_REGION

REGION Network 8: Station4/Port3 SmartLight 2 runterzaehlen
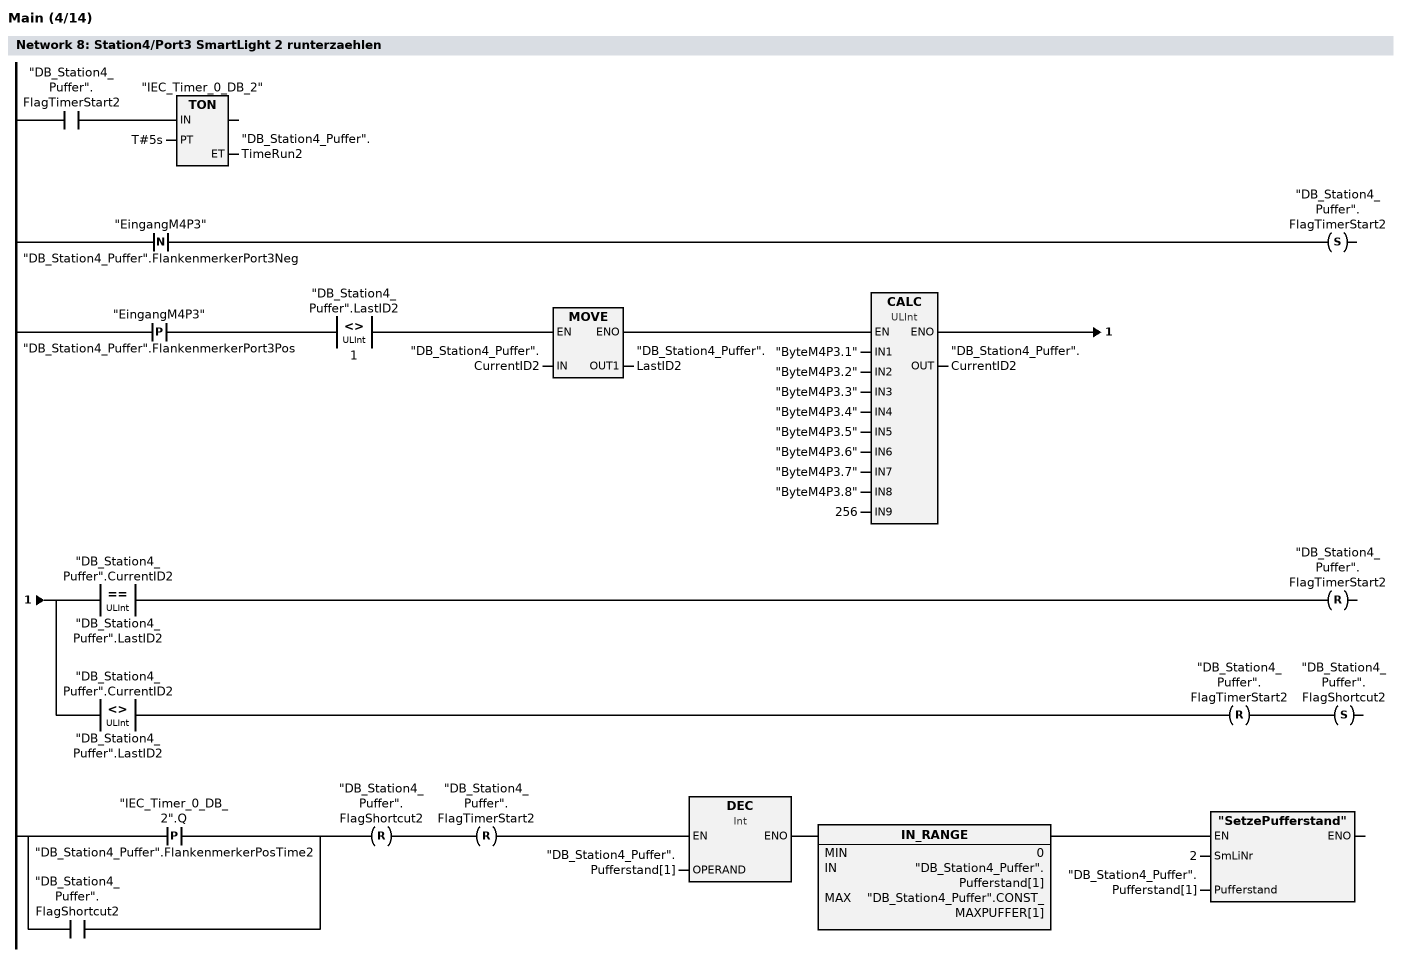
   "IEC_Timer_0_DB_2".TON(IN := "DB_Station4_Puffer".FlagTimerStart2,
                          PT := T#5s,
                          ET => "DB_Station4_Puffer".TimeRun2);
   #_w1 := NOT "EingangM4P3" AND "DB_Station4_Puffer".FlankenmerkerPort3Neg;   // falling edge of "EingangM4P3"
   "DB_Station4_Puffer".FlankenmerkerPort3Neg := "EingangM4P3";
   IF #_w1 THEN "DB_Station4_Puffer".FlagTimerStart2 := TRUE; END_IF;
   #_w2 := "EingangM4P3" AND NOT "DB_Station4_Puffer".FlankenmerkerPort3Pos;   // rising edge of "EingangM4P3"
   "DB_Station4_Puffer".FlankenmerkerPort3Pos := "EingangM4P3";
   #_w3 := #_w2 AND ("DB_Station4_Puffer".LastID2 <> 1);
   IF #_w3 THEN
       "DB_Station4_Puffer".LastID2 := "DB_Station4_Puffer".CurrentID2;
       CALC(in1 := "ByteM4P3.1",
            in2 := "ByteM4P3.2",
            in3 := "ByteM4P3.3",
            in4 := "ByteM4P3.4",
            in5 := "ByteM4P3.5",
            in6 := "ByteM4P3.6",
            in7 := "ByteM4P3.7",
            in8 := "ByteM4P3.8",
            in9 := 256,
            out => "DB_Station4_Puffer".CurrentID2);
   END_IF;
   IF #_w3 AND ("DB_Station4_Puffer".CurrentID2 = "DB_Station4_Puffer".LastID2) THEN
       "DB_Station4_Puffer".FlagTimerStart2 := FALSE;
   END_IF;
   IF #_w3 AND ("DB_Station4_Puffer".CurrentID2 <> "DB_Station4_Puffer".LastID2) THEN
       "DB_Station4_Puffer".FlagTimerStart2 := FALSE;
       "DB_Station4_Puffer".FlagShortcut2 := TRUE;
   END_IF;
   #_w4 := "IEC_Timer_0_DB_2".Q AND NOT "DB_Station4_Puffer".FlankenmerkerPosTime2;   // rising edge of "IEC_Timer_0_DB_2".Q
   "DB_Station4_Puffer".FlankenmerkerPosTime2 := "IEC_Timer_0_DB_2".Q;
   #_w5 := #_w4 OR "DB_Station4_Puffer".FlagShortcut2;
   IF #_w5 THEN
       "DB_Station4_Puffer".FlagShortcut2 := FALSE;
       "DB_Station4_Puffer".FlagTimerStart2 := FALSE;
       "DB_Station4_Puffer".Pufferstand[1] := "DB_Station4_Puffer".Pufferstand[1] - 1;
   END_IF;
   IF #_w5 AND (0 <= "DB_Station4_Puffer".Pufferstand[1]) AND ("DB_Station4_Puffer".Pufferstand[1] <= "DB_Station4_Puffer".CONST_MAXPUFFER[1]) THEN
       "SetzePufferstand"(SmLiNr := 2, Pufferstand := "DB_Station4_Puffer".Pufferstand[1]);
   END_IF;
END_REGION

REGION Network 9: Station4/Port2 schreiben (muss aktiviert werden)
   // Im Normalfall deaktivieren (Erster Schließer auf false) da nur einmalige Beschreibung der Tags (M200.0 kann als Variable zur Aktivierung verwendet werden)
   // 1. Move je nach Bedarf anpassen: 4 = kurz, 5 = lang | Schreiben in Adresse 0
   // Dokumentiert sind die Kodierungen der Header in der Beschreibung des SchreibLesekopfes
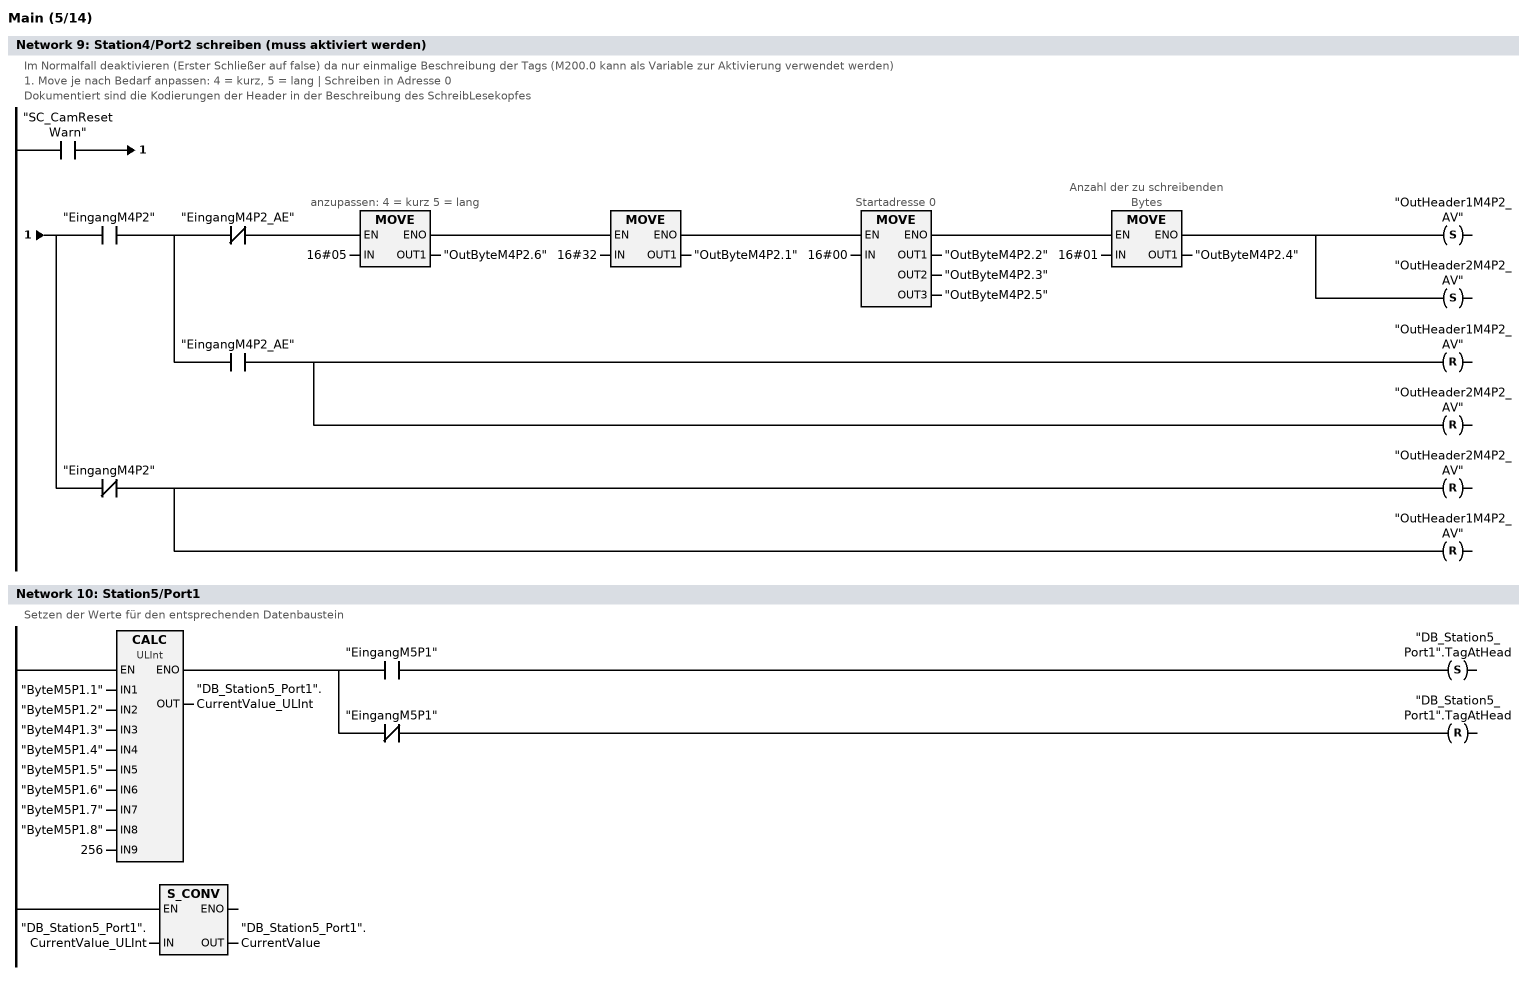
   RUNG wire#powerrail
      Contact( "SC_CamResetWarn" )
      wire#w1
      Contact( "EingangM4P2" )
      wire#w2
      I_Contact( "EingangM4P2_AE" )
      Move(in := 16#05, out1 => "OutByteM4P2.6")   // anzupassen: 4 = kurz 5 = lang
      Move(in := 16#32, out1 => "OutByteM4P2.1")
      Move(in := 16#00, out1 => "OutByteM4P2.2", out2 => "OutByteM4P2.3", out3 => "OutByteM4P2.5")   // Startadresse 0
      Move(in := 16#01, out1 => "OutByteM4P2.4")   // Anzahl der zu schreibenden Bytes
      wire#w3
      S_Coil( "OutHeader1M4P2_AV" )
   END_RUNG
   RUNG wire#w3
      S_Coil( "OutHeader2M4P2_AV" )
   END_RUNG
   RUNG wire#w2
      Contact( "EingangM4P2_AE" )
      wire#w4
      R_Coil( "OutHeader1M4P2_AV" )
   END_RUNG
   RUNG wire#w4
      R_Coil( "OutHeader2M4P2_AV" )
   END_RUNG
   RUNG wire#w1
      I_Contact( "EingangM4P2" )
      wire#w5
      R_Coil( "OutHeader2M4P2_AV" )
   END_RUNG
   RUNG wire#w5
      R_Coil( "OutHeader1M4P2_AV" )
   END_RUNG
   // the same network as SCL:
   #_w1 := "SC_CamResetWarn" AND "EingangM4P2";
   IF #_w1 AND NOT "EingangM4P2_AE" THEN
       "OutByteM4P2.6" := 16#05;   // anzupassen: 4 = kurz 5 = lang
       "OutByteM4P2.1" := 16#32;
       "OutByteM4P2.2" := 16#00;   // Startadresse 0
       "OutByteM4P2.3" := 16#00;
       "OutByteM4P2.5" := 16#00;
       "OutByteM4P2.4" := 16#01;   // Anzahl der zu schreibenden Bytes
       "OutHeader1M4P2_AV" := TRUE;
       "OutHeader2M4P2_AV" := TRUE;
   END_IF;
   IF #_w1 AND "EingangM4P2_AE" THEN
       "OutHeader1M4P2_AV" := FALSE;
       "OutHeader2M4P2_AV" := FALSE;
   END_IF;
   IF "SC_CamResetWarn" AND NOT "EingangM4P2" THEN
       "OutHeader2M4P2_AV" := FALSE;
       "OutHeader1M4P2_AV" := FALSE;
   END_IF;
END_REGION

REGION Network 10: Station5/Port1
   // Setzen der Werte für den entsprechenden Datenbaustein
   CALC(in1 := "ByteM5P1.1",
        in2 := "ByteM5P1.2",
        in3 := "ByteM4P1.3",
        in4 := "ByteM5P1.4",
        in5 := "ByteM5P1.5",
        in6 := "ByteM5P1.6",
        in7 := "ByteM5P1.7",
        in8 := "ByteM5P1.8",
        in9 := 256,
        out => "DB_Station5_Port1".CurrentValue_ULInt);
   IF "EingangM5P1" THEN "DB_Station5_Port1".TagAtHead := TRUE; END_IF;
   IF NOT "EingangM5P1" THEN "DB_Station5_Port1".TagAtHead := FALSE; END_IF;
   "DB_Station5_Port1".CurrentValue := S_CONV(IN := "DB_Station5_Port1".CurrentValue_ULInt);
END_REGION

REGION Network 11: Station6/Port1
   // Setzen der Werte für den entsprechenden Datenbaustein
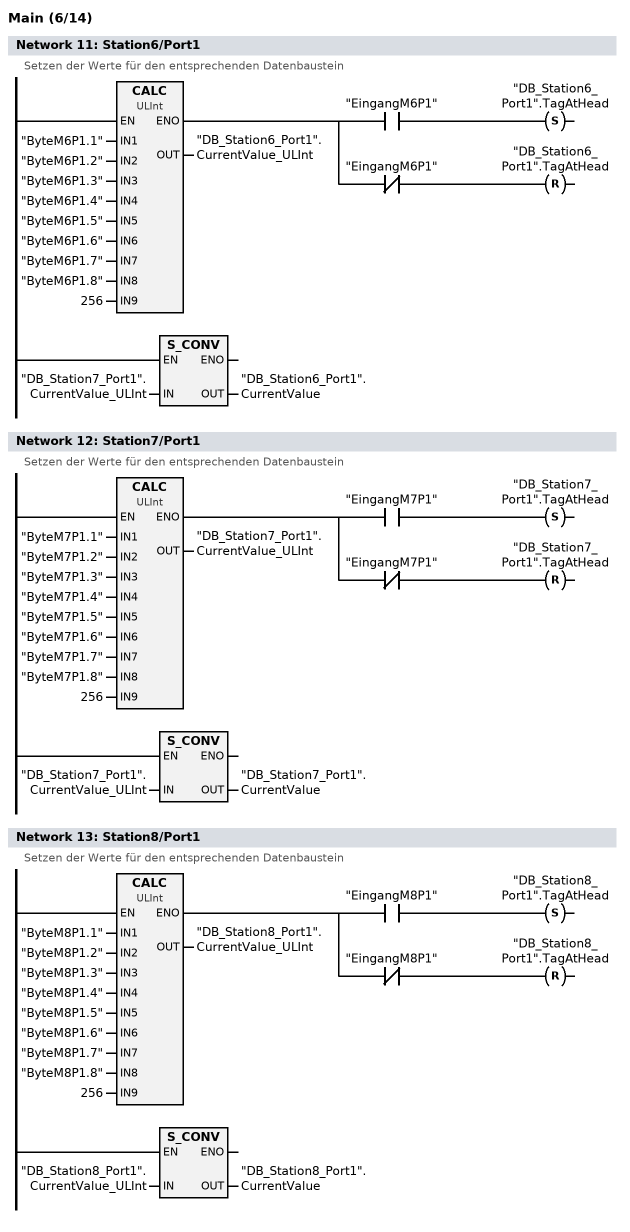
   CALC(in1 := "ByteM6P1.1",
        in2 := "ByteM6P1.2",
        in3 := "ByteM6P1.3",
        in4 := "ByteM6P1.4",
        in5 := "ByteM6P1.5",
        in6 := "ByteM6P1.6",
        in7 := "ByteM6P1.7",
        in8 := "ByteM6P1.8",
        in9 := 256,
        out => "DB_Station6_Port1".CurrentValue_ULInt);
   IF "EingangM6P1" THEN "DB_Station6_Port1".TagAtHead := TRUE; END_IF;
   IF NOT "EingangM6P1" THEN "DB_Station6_Port1".TagAtHead := FALSE; END_IF;
   "DB_Station6_Port1".CurrentValue := S_CONV(IN := "DB_Station7_Port1".CurrentValue_ULInt);
END_REGION

REGION Network 12: Station7/Port1
   // Setzen der Werte für den entsprechenden Datenbaustein
   CALC(in1 := "ByteM7P1.1",
        in2 := "ByteM7P1.2",
        in3 := "ByteM7P1.3",
        in4 := "ByteM7P1.4",
        in5 := "ByteM7P1.5",
        in6 := "ByteM7P1.6",
        in7 := "ByteM7P1.7",
        in8 := "ByteM7P1.8",
        in9 := 256,
        out => "DB_Station7_Port1".CurrentValue_ULInt);
   IF "EingangM7P1" THEN "DB_Station7_Port1".TagAtHead := TRUE; END_IF;
   IF NOT "EingangM7P1" THEN "DB_Station7_Port1".TagAtHead := FALSE; END_IF;
   "DB_Station7_Port1".CurrentValue := S_CONV(IN := "DB_Station7_Port1".CurrentValue_ULInt);
END_REGION

REGION Network 13: Station8/Port1
   // Setzen der Werte für den entsprechenden Datenbaustein
   CALC(in1 := "ByteM8P1.1",
        in2 := "ByteM8P1.2",
        in3 := "ByteM8P1.3",
        in4 := "ByteM8P1.4",
        in5 := "ByteM8P1.5",
        in6 := "ByteM8P1.6",
        in7 := "ByteM8P1.7",
        in8 := "ByteM8P1.8",
        in9 := 256,
        out => "DB_Station8_Port1".CurrentValue_ULInt);
   IF "EingangM8P1" THEN "DB_Station8_Port1".TagAtHead := TRUE; END_IF;
   IF NOT "EingangM8P1" THEN "DB_Station8_Port1".TagAtHead := FALSE; END_IF;
   "DB_Station8_Port1".CurrentValue := S_CONV(IN := "DB_Station8_Port1".CurrentValue_ULInt);
END_REGION

REGION Network 14: Station8/Port2
   // Setzen der Werte für den entsprechenden Datenbaustein
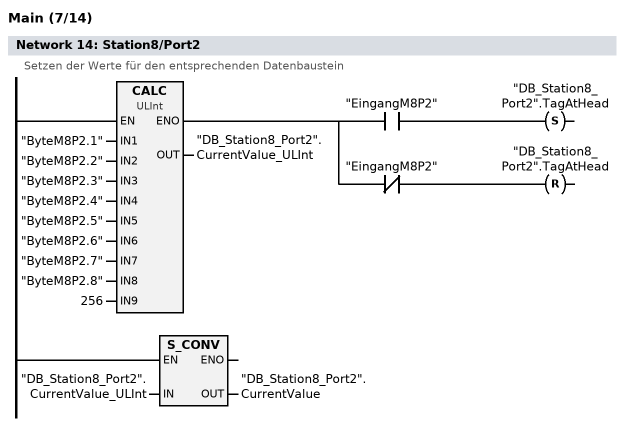
   CALC(in1 := "ByteM8P2.1",
        in2 := "ByteM8P2.2",
        in3 := "ByteM8P2.3",
        in4 := "ByteM8P2.4",
        in5 := "ByteM8P2.5",
        in6 := "ByteM8P2.6",
        in7 := "ByteM8P2.7",
        in8 := "ByteM8P2.8",
        in9 := 256,
        out => "DB_Station8_Port2".CurrentValue_ULInt);
   IF "EingangM8P2" THEN "DB_Station8_Port2".TagAtHead := TRUE; END_IF;
   IF NOT "EingangM8P2" THEN "DB_Station8_Port2".TagAtHead := FALSE; END_IF;
   "DB_Station8_Port2".CurrentValue := S_CONV(IN := "DB_Station8_Port2".CurrentValue_ULInt);
END_REGION

REGION Network 15: Station8/SmartCamera
   // Das Kommando Switch Application darf nur ausgeführt werden wenn die Kamera nicht läuft (Cam-Running = false)
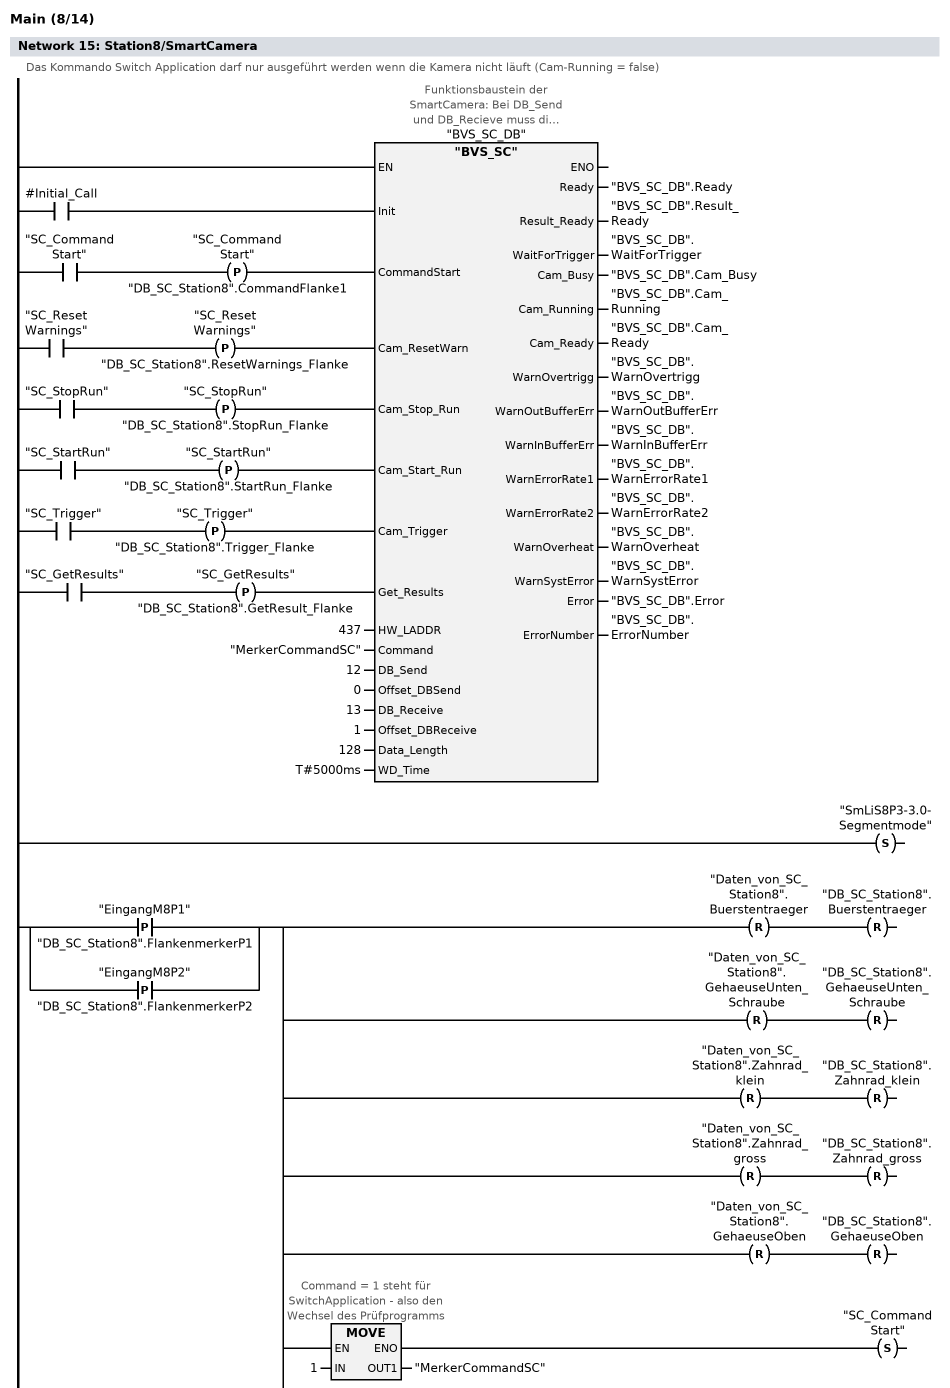
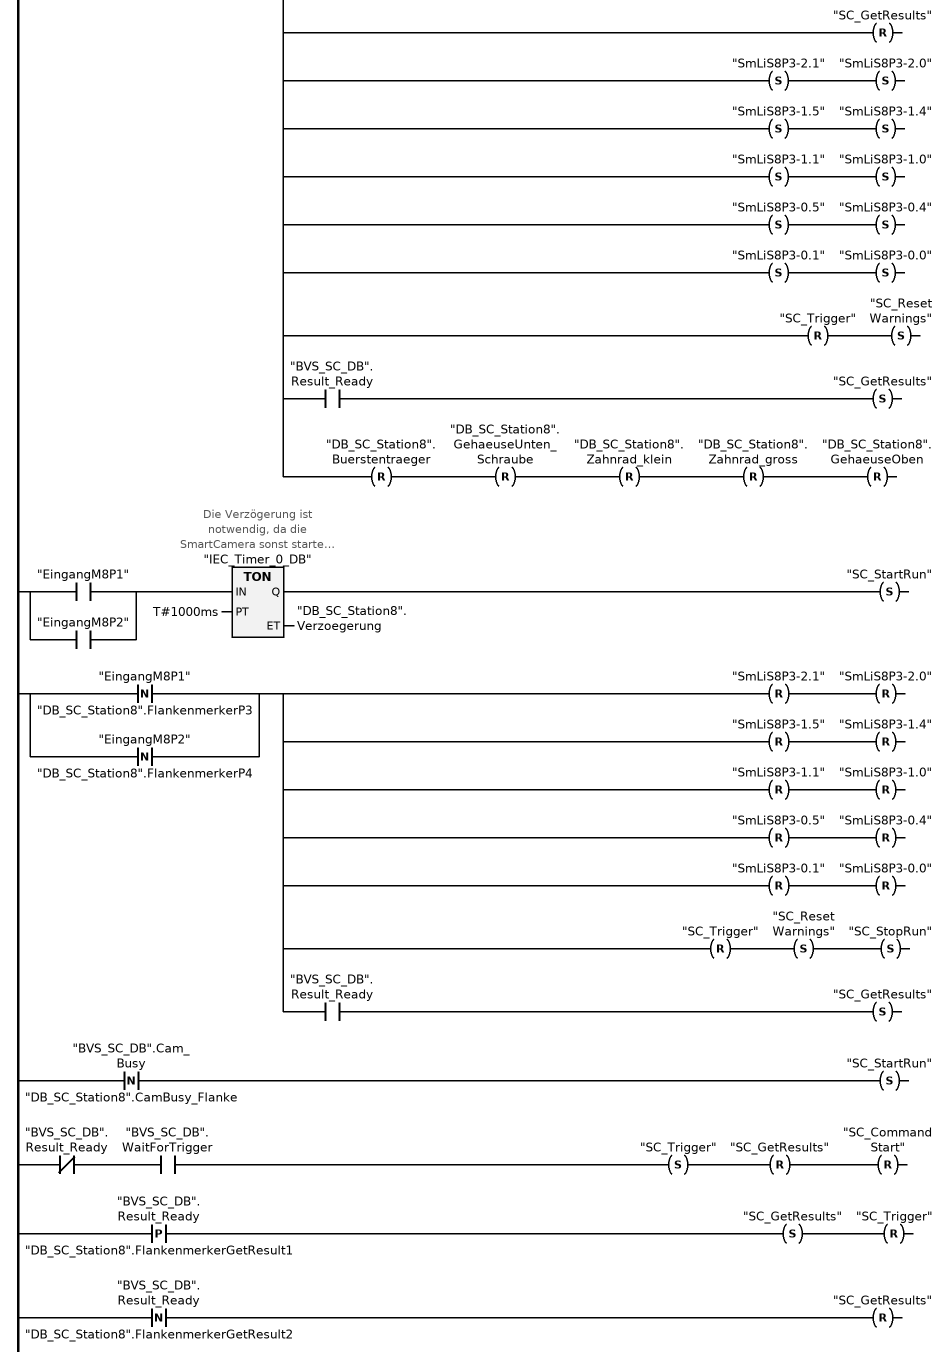
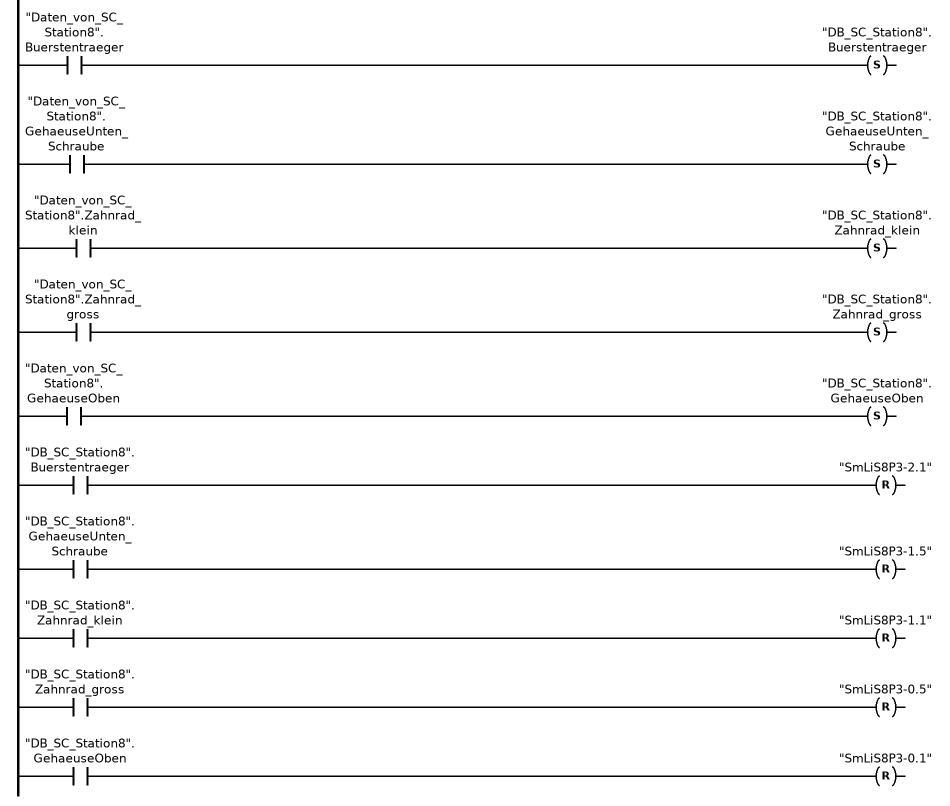
   #_w1 := "SC_CommandStart";
   "SC_CommandStart" := #_w1 AND NOT "DB_SC_Station8".CommandFlanke1;   // rising edge
   "DB_SC_Station8".CommandFlanke1 := #_w1;
   #_w2 := "SC_ResetWarnings";
   "SC_ResetWarnings" := #_w2 AND NOT "DB_SC_Station8".ResetWarnings_Flanke;   // rising edge
   "DB_SC_Station8".ResetWarnings_Flanke := #_w2;
   #_w3 := "SC_StopRun";
   "SC_StopRun" := #_w3 AND NOT "DB_SC_Station8".StopRun_Flanke;   // rising edge
   "DB_SC_Station8".StopRun_Flanke := #_w3;
   #_w4 := "SC_StartRun";
   "SC_StartRun" := #_w4 AND NOT "DB_SC_Station8".StartRun_Flanke;   // rising edge
   "DB_SC_Station8".StartRun_Flanke := #_w4;
   #_w5 := "SC_Trigger";
   "SC_Trigger" := #_w5 AND NOT "DB_SC_Station8".Trigger_Flanke;   // rising edge
   "DB_SC_Station8".Trigger_Flanke := #_w5;
   #_w6 := "SC_GetResults";
   "SC_GetResults" := #_w6 AND NOT "DB_SC_Station8".GetResult_Flanke;   // rising edge
   "DB_SC_Station8".GetResult_Flanke := #_w6;
   "BVS_SC_DB"(Init := #Initial_Call,   // "BVS_SC": Funktionsbaustein der SmartCamera: Bei DB_Send und DB_Recieve muss die Nummer des verwendeten Datenbausteins angegeben werden.
               CommandStart := #_w1,
               Cam_ResetWarn := #_w2,
               Cam_Stop_Run := #_w3,
               Cam_Start_Run := #_w4,
               Cam_Trigger := #_w5,
               Get_Results := #_w6,
               HW_LADDR := 437,
               Command := "MerkerCommandSC",
               DB_Send := 12,
               Offset_DBSend := 0,
               DB_Receive := 13,
               Offset_DBReceive := 1,
               Data_Length := 128,
               WD_Time := T#5000ms,
               Ready => "BVS_SC_DB".Ready,
               Result_Ready => "BVS_SC_DB".Result_Ready,
               WaitForTrigger => "BVS_SC_DB".WaitForTrigger,
               Cam_Busy => "BVS_SC_DB".Cam_Busy,
               Cam_Running => "BVS_SC_DB".Cam_Running,
               Cam_Ready => "BVS_SC_DB".Cam_Ready,
               WarnOvertrigg => "BVS_SC_DB".WarnOvertrigg,
               WarnOutBufferErr => "BVS_SC_DB".WarnOutBufferErr,
               WarnInBufferErr => "BVS_SC_DB".WarnInBufferErr,
               WarnErrorRate1 => "BVS_SC_DB".WarnErrorRate1,
               WarnErrorRate2 => "BVS_SC_DB".WarnErrorRate2,
               WarnOverheat => "BVS_SC_DB".WarnOverheat,
               WarnSystError => "BVS_SC_DB".WarnSystError,
               Error => "BVS_SC_DB".Error,
               ErrorNumber => "BVS_SC_DB".ErrorNumber);
   "SmLiS8P3-3.0-Segmentmode" := TRUE;
   #_w7 := "EingangM8P1" AND NOT "DB_SC_Station8".FlankenmerkerP1;   // rising edge of "EingangM8P1"
   "DB_SC_Station8".FlankenmerkerP1 := "EingangM8P1";
   #_w8 := "EingangM8P2" AND NOT "DB_SC_Station8".FlankenmerkerP2;   // rising edge of "EingangM8P2"
   "DB_SC_Station8".FlankenmerkerP2 := "EingangM8P2";
   #_w9 := #_w7 OR #_w8;
   IF #_w9 THEN
       "Daten_von_SC_Station8".Buerstentraeger := FALSE;
       "DB_SC_Station8".Buerstentraeger := FALSE;
       "Daten_von_SC_Station8".GehaeuseUnten_Schraube := FALSE;
       "DB_SC_Station8".GehaeuseUnten_Schraube := FALSE;
       "Daten_von_SC_Station8".Zahnrad_klein := FALSE;
       "DB_SC_Station8".Zahnrad_klein := FALSE;
       "Daten_von_SC_Station8".Zahnrad_gross := FALSE;
       "DB_SC_Station8".Zahnrad_gross := FALSE;
       "Daten_von_SC_Station8".GehaeuseOben := FALSE;
       "DB_SC_Station8".GehaeuseOben := FALSE;
       "MerkerCommandSC" := 1;   // Command = 1 steht für SwitchApplication - also den Wechsel des Prüfprogramms
       "SC_CommandStart" := TRUE;
       "SC_GetResults" := FALSE;
       "SmLiS8P3-2.1" := TRUE;
       "SmLiS8P3-2.0" := TRUE;
       "SmLiS8P3-1.5" := TRUE;
       "SmLiS8P3-1.4" := TRUE;
       "SmLiS8P3-1.1" := TRUE;
       "SmLiS8P3-1.0" := TRUE;
       "SmLiS8P3-0.5" := TRUE;
       "SmLiS8P3-0.4" := TRUE;
       "SmLiS8P3-0.1" := TRUE;
       "SmLiS8P3-0.0" := TRUE;
       "SC_Trigger" := FALSE;
       "SC_ResetWarnings" := TRUE;
   END_IF;
   IF #_w9 AND "BVS_SC_DB".Result_Ready THEN "SC_GetResults" := TRUE; END_IF;
   IF #_w9 THEN
       "DB_SC_Station8".Buerstentraeger := FALSE;
       "DB_SC_Station8".GehaeuseUnten_Schraube := FALSE;
       "DB_SC_Station8".Zahnrad_klein := FALSE;
       "DB_SC_Station8".Zahnrad_gross := FALSE;
       "DB_SC_Station8".GehaeuseOben := FALSE;
   END_IF;
   "IEC_Timer_0_DB".TON(IN := "EingangM8P1" OR "EingangM8P2",   // Die Verzögerung ist notwendig, da die SmartCamera sonst startet bevor der Wechsel des Prüfprogramms ausgelöst wird. Dies führt zu einem Fehler.
                        PT := T#1000ms,
                        ET => "DB_SC_Station8".Verzoegerung);
   IF "IEC_Timer_0_DB".Q THEN "SC_StartRun" := TRUE; END_IF;
   #_w10 := NOT "EingangM8P1" AND "DB_SC_Station8".FlankenmerkerP3;   // falling edge of "EingangM8P1"
   "DB_SC_Station8".FlankenmerkerP3 := "EingangM8P1";
   #_w11 := NOT "EingangM8P2" AND "DB_SC_Station8".FlankenmerkerP4;   // falling edge of "EingangM8P2"
   "DB_SC_Station8".FlankenmerkerP4 := "EingangM8P2";
   #_w12 := #_w10 OR #_w11;
   IF #_w12 THEN
       "SmLiS8P3-2.1" := FALSE;
       "SmLiS8P3-2.0" := FALSE;
       "SmLiS8P3-1.5" := FALSE;
       "SmLiS8P3-1.4" := FALSE;
       "SmLiS8P3-1.1" := FALSE;
       "SmLiS8P3-1.0" := FALSE;
       "SmLiS8P3-0.5" := FALSE;
       "SmLiS8P3-0.4" := FALSE;
       "SmLiS8P3-0.1" := FALSE;
       "SmLiS8P3-0.0" := FALSE;
       "SC_Trigger" := FALSE;
       "SC_ResetWarnings" := TRUE;
       "SC_StopRun" := TRUE;
   END_IF;
   IF #_w12 AND "BVS_SC_DB".Result_Ready THEN "SC_GetResults" := TRUE; END_IF;
   #_w13 := NOT "BVS_SC_DB".Cam_Busy AND "DB_SC_Station8".CamBusy_Flanke;   // falling edge of "BVS_SC_DB".Cam_Busy
   "DB_SC_Station8".CamBusy_Flanke := "BVS_SC_DB".Cam_Busy;
   IF #_w13 THEN "SC_StartRun" := TRUE; END_IF;
   IF NOT "BVS_SC_DB".Result_Ready AND "BVS_SC_DB".WaitForTrigger THEN
       "SC_Trigger" := TRUE;
       "SC_GetResults" := FALSE;
       "SC_CommandStart" := FALSE;
   END_IF;
   #_w14 := "BVS_SC_DB".Result_Ready AND NOT "DB_SC_Station8".FlankenmerkerGetResult1;   // rising edge of "BVS_SC_DB".Result_Ready
   "DB_SC_Station8".FlankenmerkerGetResult1 := "BVS_SC_DB".Result_Ready;
   IF #_w14 THEN
       "SC_GetResults" := TRUE;
       "SC_Trigger" := FALSE;
   END_IF;
   #_w15 := NOT "BVS_SC_DB".Result_Ready AND "DB_SC_Station8".FlankenmerkerGetResult2;   // falling edge of "BVS_SC_DB".Result_Ready
   "DB_SC_Station8".FlankenmerkerGetResult2 := "BVS_SC_DB".Result_Ready;
   IF #_w15 THEN "SC_GetResults" := FALSE; END_IF;
   IF "Daten_von_SC_Station8".Buerstentraeger THEN "DB_SC_Station8".Buerstentraeger := TRUE; END_IF;
   IF "Daten_von_SC_Station8".GehaeuseUnten_Schraube THEN
       "DB_SC_Station8".GehaeuseUnten_Schraube := TRUE;
   END_IF;
   IF "Daten_von_SC_Station8".Zahnrad_klein THEN "DB_SC_Station8".Zahnrad_klein := TRUE; END_IF;
   IF "Daten_von_SC_Station8".Zahnrad_gross THEN "DB_SC_Station8".Zahnrad_gross := TRUE; END_IF;
   IF "Daten_von_SC_Station8".GehaeuseOben THEN "DB_SC_Station8".GehaeuseOben := TRUE; END_IF;
   IF "DB_SC_Station8".Buerstentraeger THEN "SmLiS8P3-2.1" := FALSE; END_IF;
   IF "DB_SC_Station8".GehaeuseUnten_Schraube THEN "SmLiS8P3-1.5" := FALSE; END_IF;
   IF "DB_SC_Station8".Zahnrad_klein THEN "SmLiS8P3-1.1" := FALSE; END_IF;
   IF "DB_SC_Station8".Zahnrad_gross THEN "SmLiS8P3-0.5" := FALSE; END_IF;
   IF "DB_SC_Station8".GehaeuseOben THEN "SmLiS8P3-0.1" := FALSE; END_IF;
END_REGION

REGION Network 16: Station9/Port1
   // Setzen der Werte für den entsprechenden Datenbaustein
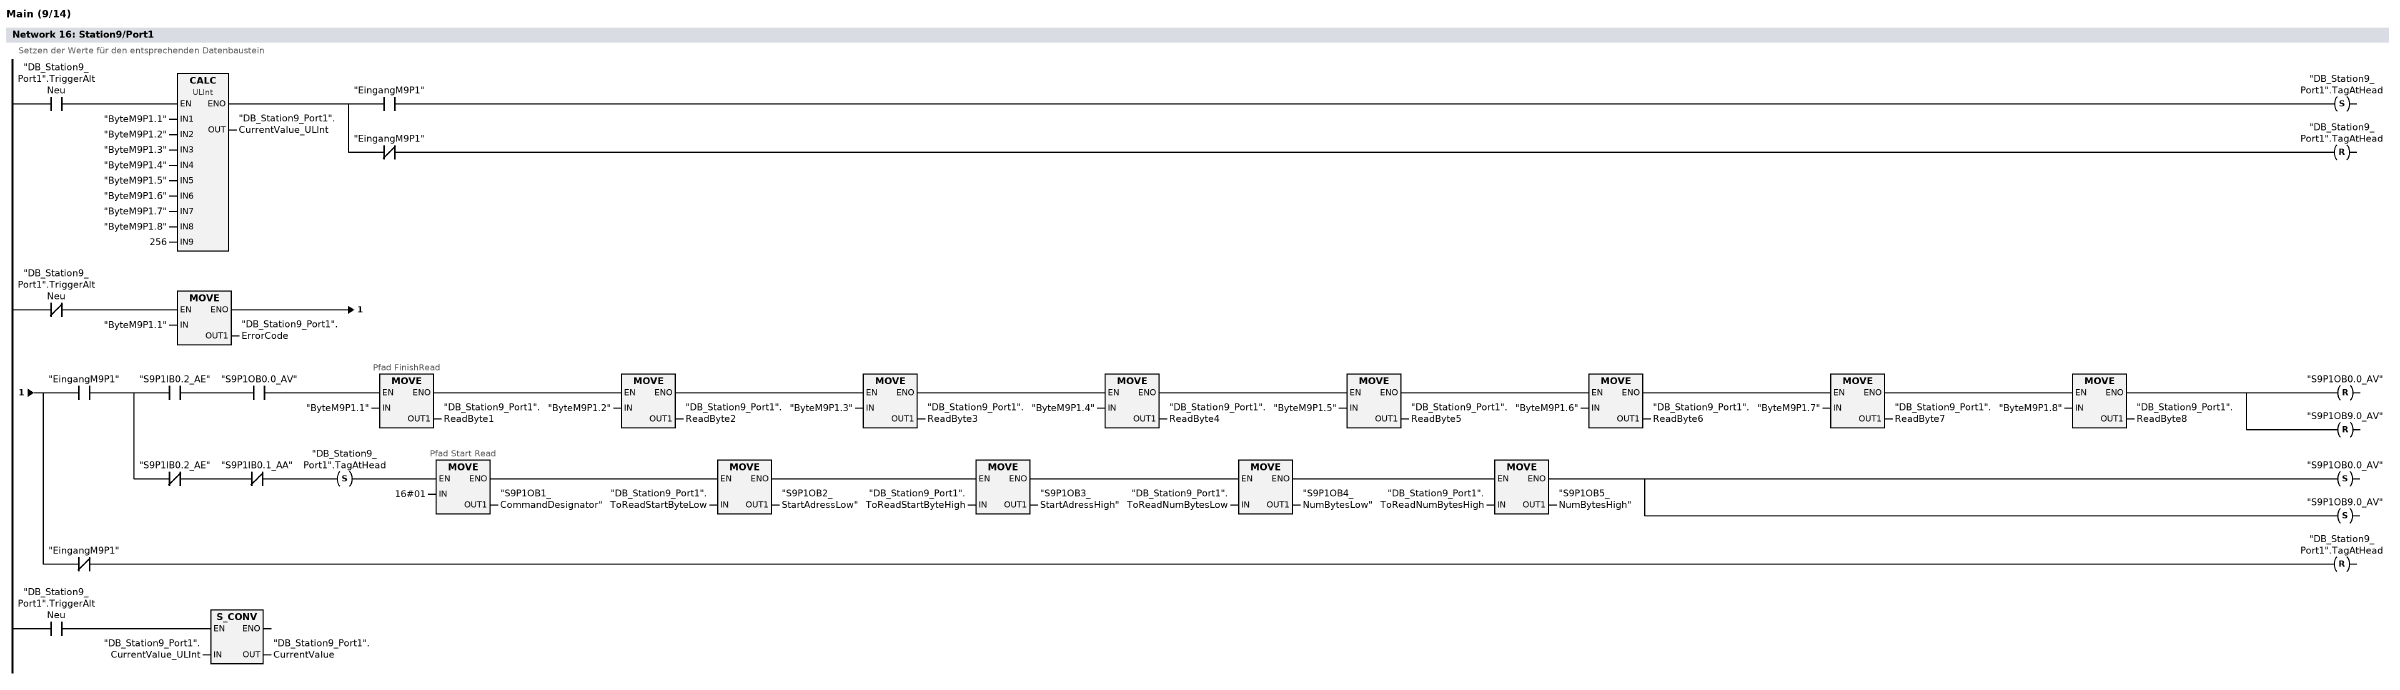
   #_w1 := "DB_Station9_Port1".TriggerAltNeu;
   IF #_w1 THEN
       CALC(in1 := "ByteM9P1.1",
            in2 := "ByteM9P1.2",
            in3 := "ByteM9P1.3",
            in4 := "ByteM9P1.4",
            in5 := "ByteM9P1.5",
            in6 := "ByteM9P1.6",
            in7 := "ByteM9P1.7",
            in8 := "ByteM9P1.8",
            in9 := 256,
            out => "DB_Station9_Port1".CurrentValue_ULInt);
   END_IF;
   IF #_w1 AND "EingangM9P1" THEN "DB_Station9_Port1".TagAtHead := TRUE; END_IF;
   IF #_w1 AND NOT "EingangM9P1" THEN "DB_Station9_Port1".TagAtHead := FALSE; END_IF;
   #_w2 := NOT "DB_Station9_Port1".TriggerAltNeu;
   IF #_w2 THEN "DB_Station9_Port1".ErrorCode := "ByteM9P1.1"; END_IF;
   #_w3 := #_w2 AND "EingangM9P1";
   IF #_w3 AND "S9P1IB0.2_AE" AND "S9P1OB0.0_AV" THEN
       "DB_Station9_Port1".ReadByte1 := "ByteM9P1.1";   // Pfad FinishRead
       "DB_Station9_Port1".ReadByte2 := "ByteM9P1.2";
       "DB_Station9_Port1".ReadByte3 := "ByteM9P1.3";
       "DB_Station9_Port1".ReadByte4 := "ByteM9P1.4";
       "DB_Station9_Port1".ReadByte5 := "ByteM9P1.5";
       "DB_Station9_Port1".ReadByte6 := "ByteM9P1.6";
       "DB_Station9_Port1".ReadByte7 := "ByteM9P1.7";
       "DB_Station9_Port1".ReadByte8 := "ByteM9P1.8";
   END_IF;
   #_w4 := #_w3 AND "S9P1IB0.2_AE" AND "S9P1OB0.0_AV";
   IF #_w4 THEN
       "S9P1OB0.0_AV" := FALSE;
       "S9P1OB9.0_AV" := FALSE;
   END_IF;
   IF #_w3 AND NOT "S9P1IB0.2_AE" AND NOT "S9P1IB0.1_AA" THEN
       "DB_Station9_Port1".TagAtHead := TRUE;
       "S9P1OB1_CommandDesignator" := 16#01;   // Pfad Start Read
       "S9P1OB2_StartAdressLow" := "DB_Station9_Port1".ToReadStartByteLow;
       "S9P1OB3_StartAdressHigh" := "DB_Station9_Port1".ToReadStartByteHigh;
       "S9P1OB4_NumBytesLow" := "DB_Station9_Port1".ToReadNumBytesLow;
       "S9P1OB5_NumBytesHigh" := "DB_Station9_Port1".ToReadNumBytesHigh;
       "S9P1OB0.0_AV" := TRUE;
       "S9P1OB9.0_AV" := TRUE;
   END_IF;
   IF #_w2 AND NOT "EingangM9P1" THEN "DB_Station9_Port1".TagAtHead := FALSE; END_IF;
   IF "DB_Station9_Port1".TriggerAltNeu THEN
       "DB_Station9_Port1".CurrentValue := S_CONV(IN := "DB_Station9_Port1".CurrentValue_ULInt);
   END_IF;
END_REGION

REGION Network 17: Station9/Port2
   // Setzen der Werte für den entsprechenden Datenbaustein
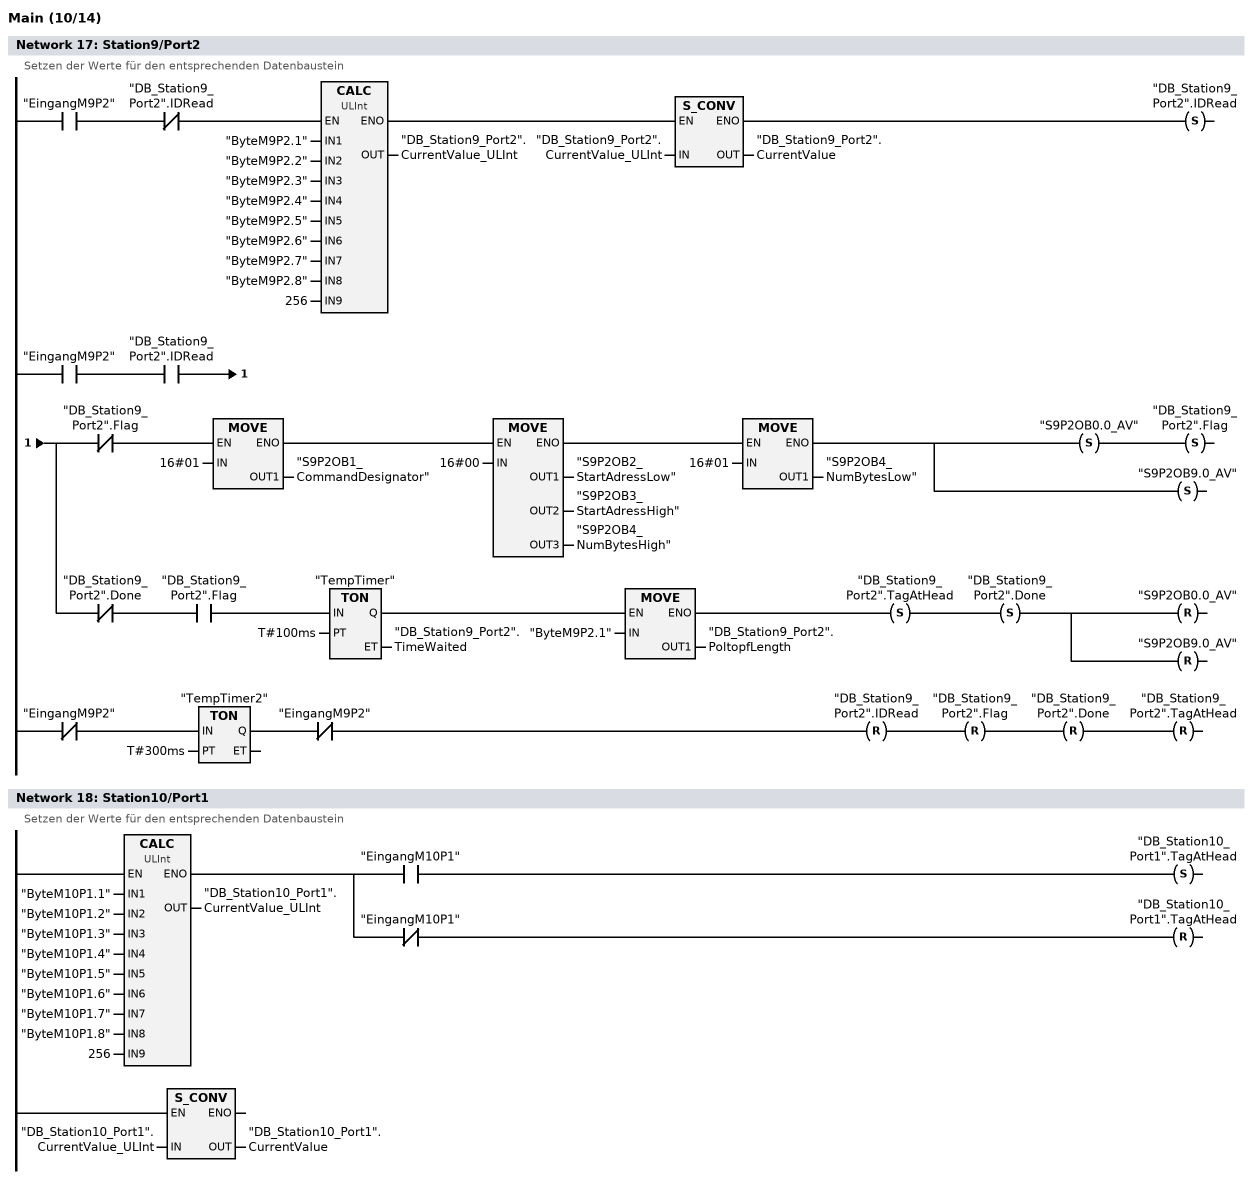
   #_w1 := "EingangM9P2" AND NOT "DB_Station9_Port2".IDRead;
   IF #_w1 THEN
       CALC(in1 := "ByteM9P2.1",
            in2 := "ByteM9P2.2",
            in3 := "ByteM9P2.3",
            in4 := "ByteM9P2.4",
            in5 := "ByteM9P2.5",
            in6 := "ByteM9P2.6",
            in7 := "ByteM9P2.7",
            in8 := "ByteM9P2.8",
            in9 := 256,
            out => "DB_Station9_Port2".CurrentValue_ULInt);
       "DB_Station9_Port2".CurrentValue := S_CONV(IN := "DB_Station9_Port2".CurrentValue_ULInt);
       "DB_Station9_Port2".IDRead := TRUE;
   END_IF;
   #_w2 := "EingangM9P2" AND "DB_Station9_Port2".IDRead;
   IF #_w2 AND NOT "DB_Station9_Port2".Flag THEN
       "S9P2OB1_CommandDesignator" := 16#01;
       "S9P2OB2_StartAdressLow" := 16#00;
       "S9P2OB3_StartAdressHigh" := 16#00;
       "S9P2OB4_NumBytesHigh" := 16#00;
       "S9P2OB4_NumBytesLow" := 16#01;
       "S9P2OB0.0_AV" := TRUE;
   END_IF;
   #_w3 := #_w2 AND NOT "DB_Station9_Port2".Flag;
   IF #_w3 THEN
       "DB_Station9_Port2".Flag := TRUE;
       "S9P2OB9.0_AV" := TRUE;
   END_IF;
   "TempTimer".TON(IN := #_w2 AND NOT "DB_Station9_Port2".Done AND "DB_Station9_Port2".Flag,
                   PT := T#100ms,
                   ET => "DB_Station9_Port2".TimeWaited);
   IF "TempTimer".Q THEN
       "DB_Station9_Port2".PoltopfLength := "ByteM9P2.1";
       "DB_Station9_Port2".TagAtHead := TRUE;
       "DB_Station9_Port2".Done := TRUE;
       "S9P2OB0.0_AV" := FALSE;
       "S9P2OB9.0_AV" := FALSE;
   END_IF;
   "TempTimer2".TON(IN := NOT "EingangM9P2", PT := T#300ms);
   IF "TempTimer2".Q AND NOT "EingangM9P2" THEN
       "DB_Station9_Port2".IDRead := FALSE;
       "DB_Station9_Port2".Flag := FALSE;
       "DB_Station9_Port2".Done := FALSE;
       "DB_Station9_Port2".TagAtHead := FALSE;
   END_IF;
END_REGION

REGION Network 18: Station10/Port1
   // Setzen der Werte für den entsprechenden Datenbaustein
   CALC(in1 := "ByteM10P1.1",
        in2 := "ByteM10P1.2",
        in3 := "ByteM10P1.3",
        in4 := "ByteM10P1.4",
        in5 := "ByteM10P1.5",
        in6 := "ByteM10P1.6",
        in7 := "ByteM10P1.7",
        in8 := "ByteM10P1.8",
        in9 := 256,
        out => "DB_Station10_Port1".CurrentValue_ULInt);
   IF "EingangM10P1" THEN "DB_Station10_Port1".TagAtHead := TRUE; END_IF;
   IF NOT "EingangM10P1" THEN "DB_Station10_Port1".TagAtHead := FALSE; END_IF;
   "DB_Station10_Port1".CurrentValue := S_CONV(IN := "DB_Station10_Port1".CurrentValue_ULInt);
END_REGION

REGION Network 19: Station11/Port1
   // Setzen der Werte für den entsprechenden Datenbaustein
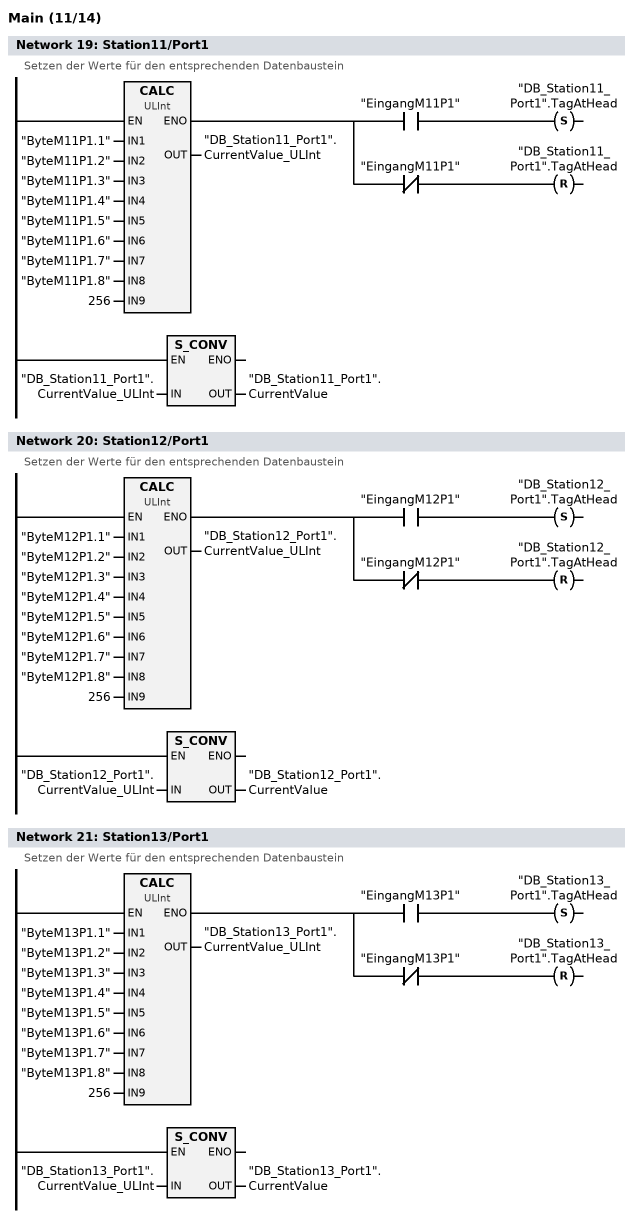
   CALC(in1 := "ByteM11P1.1",
        in2 := "ByteM11P1.2",
        in3 := "ByteM11P1.3",
        in4 := "ByteM11P1.4",
        in5 := "ByteM11P1.5",
        in6 := "ByteM11P1.6",
        in7 := "ByteM11P1.7",
        in8 := "ByteM11P1.8",
        in9 := 256,
        out => "DB_Station11_Port1".CurrentValue_ULInt);
   IF "EingangM11P1" THEN "DB_Station11_Port1".TagAtHead := TRUE; END_IF;
   IF NOT "EingangM11P1" THEN "DB_Station11_Port1".TagAtHead := FALSE; END_IF;
   "DB_Station11_Port1".CurrentValue := S_CONV(IN := "DB_Station11_Port1".CurrentValue_ULInt);
END_REGION

REGION Network 20: Station12/Port1
   // Setzen der Werte für den entsprechenden Datenbaustein
   CALC(in1 := "ByteM12P1.1",
        in2 := "ByteM12P1.2",
        in3 := "ByteM12P1.3",
        in4 := "ByteM12P1.4",
        in5 := "ByteM12P1.5",
        in6 := "ByteM12P1.6",
        in7 := "ByteM12P1.7",
        in8 := "ByteM12P1.8",
        in9 := 256,
        out => "DB_Station12_Port1".CurrentValue_ULInt);
   IF "EingangM12P1" THEN "DB_Station12_Port1".TagAtHead := TRUE; END_IF;
   IF NOT "EingangM12P1" THEN "DB_Station12_Port1".TagAtHead := FALSE; END_IF;
   "DB_Station12_Port1".CurrentValue := S_CONV(IN := "DB_Station12_Port1".CurrentValue_ULInt);
END_REGION

REGION Network 21: Station13/Port1
   // Setzen der Werte für den entsprechenden Datenbaustein
   CALC(in1 := "ByteM13P1.1",
        in2 := "ByteM13P1.2",
        in3 := "ByteM13P1.3",
        in4 := "ByteM13P1.4",
        in5 := "ByteM13P1.5",
        in6 := "ByteM13P1.6",
        in7 := "ByteM13P1.7",
        in8 := "ByteM13P1.8",
        in9 := 256,
        out => "DB_Station13_Port1".CurrentValue_ULInt);
   IF "EingangM13P1" THEN "DB_Station13_Port1".TagAtHead := TRUE; END_IF;
   IF NOT "EingangM13P1" THEN "DB_Station13_Port1".TagAtHead := FALSE; END_IF;
   "DB_Station13_Port1".CurrentValue := S_CONV(IN := "DB_Station13_Port1".CurrentValue_ULInt);
END_REGION

REGION Network 22: Station15/Port1
   // Setzen der Werte für den entsprechenden Datenbaustein
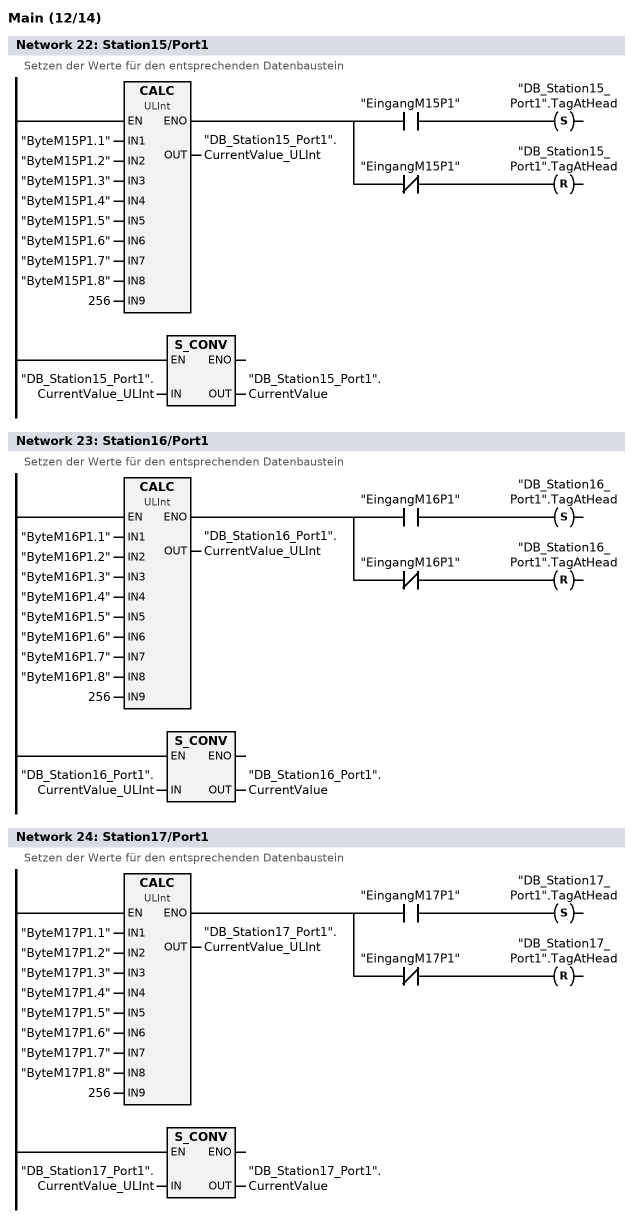
   CALC(in1 := "ByteM15P1.1",
        in2 := "ByteM15P1.2",
        in3 := "ByteM15P1.3",
        in4 := "ByteM15P1.4",
        in5 := "ByteM15P1.5",
        in6 := "ByteM15P1.6",
        in7 := "ByteM15P1.7",
        in8 := "ByteM15P1.8",
        in9 := 256,
        out => "DB_Station15_Port1".CurrentValue_ULInt);
   IF "EingangM15P1" THEN "DB_Station15_Port1".TagAtHead := TRUE; END_IF;
   IF NOT "EingangM15P1" THEN "DB_Station15_Port1".TagAtHead := FALSE; END_IF;
   "DB_Station15_Port1".CurrentValue := S_CONV(IN := "DB_Station15_Port1".CurrentValue_ULInt);
END_REGION

REGION Network 23: Station16/Port1
   // Setzen der Werte für den entsprechenden Datenbaustein
   CALC(in1 := "ByteM16P1.1",
        in2 := "ByteM16P1.2",
        in3 := "ByteM16P1.3",
        in4 := "ByteM16P1.4",
        in5 := "ByteM16P1.5",
        in6 := "ByteM16P1.6",
        in7 := "ByteM16P1.7",
        in8 := "ByteM16P1.8",
        in9 := 256,
        out => "DB_Station16_Port1".CurrentValue_ULInt);
   IF "EingangM16P1" THEN "DB_Station16_Port1".TagAtHead := TRUE; END_IF;
   IF NOT "EingangM16P1" THEN "DB_Station16_Port1".TagAtHead := FALSE; END_IF;
   "DB_Station16_Port1".CurrentValue := S_CONV(IN := "DB_Station16_Port1".CurrentValue_ULInt);
END_REGION

REGION Network 24: Station17/Port1
   // Setzen der Werte für den entsprechenden Datenbaustein
   CALC(in1 := "ByteM17P1.1",
        in2 := "ByteM17P1.2",
        in3 := "ByteM17P1.3",
        in4 := "ByteM17P1.4",
        in5 := "ByteM17P1.5",
        in6 := "ByteM17P1.6",
        in7 := "ByteM17P1.7",
        in8 := "ByteM17P1.8",
        in9 := 256,
        out => "DB_Station17_Port1".CurrentValue_ULInt);
   IF "EingangM17P1" THEN "DB_Station17_Port1".TagAtHead := TRUE; END_IF;
   IF NOT "EingangM17P1" THEN "DB_Station17_Port1".TagAtHead := FALSE; END_IF;
   "DB_Station17_Port1".CurrentValue := S_CONV(IN := "DB_Station17_Port1".CurrentValue_ULInt);
END_REGION

REGION Network 25: Station19/Port1
   // Setzen der Werte für den entsprechenden Datenbaustein
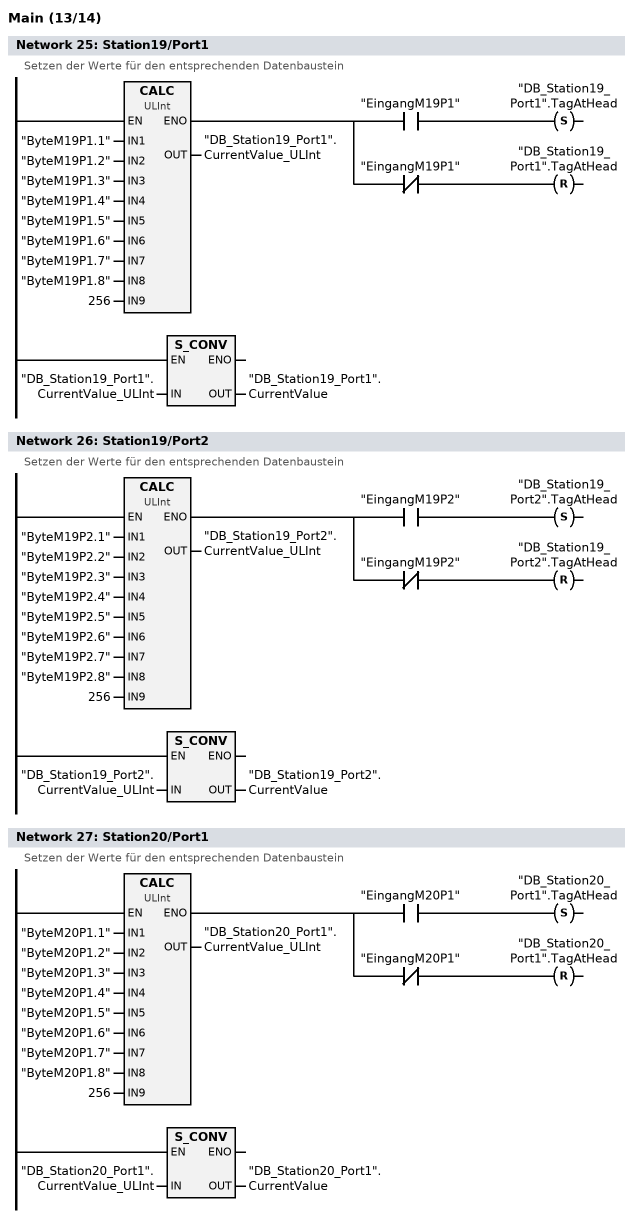
   CALC(in1 := "ByteM19P1.1",
        in2 := "ByteM19P1.2",
        in3 := "ByteM19P1.3",
        in4 := "ByteM19P1.4",
        in5 := "ByteM19P1.5",
        in6 := "ByteM19P1.6",
        in7 := "ByteM19P1.7",
        in8 := "ByteM19P1.8",
        in9 := 256,
        out => "DB_Station19_Port1".CurrentValue_ULInt);
   IF "EingangM19P1" THEN "DB_Station19_Port1".TagAtHead := TRUE; END_IF;
   IF NOT "EingangM19P1" THEN "DB_Station19_Port1".TagAtHead := FALSE; END_IF;
   "DB_Station19_Port1".CurrentValue := S_CONV(IN := "DB_Station19_Port1".CurrentValue_ULInt);
END_REGION

REGION Network 26: Station19/Port2
   // Setzen der Werte für den entsprechenden Datenbaustein
   CALC(in1 := "ByteM19P2.1",
        in2 := "ByteM19P2.2",
        in3 := "ByteM19P2.3",
        in4 := "ByteM19P2.4",
        in5 := "ByteM19P2.5",
        in6 := "ByteM19P2.6",
        in7 := "ByteM19P2.7",
        in8 := "ByteM19P2.8",
        in9 := 256,
        out => "DB_Station19_Port2".CurrentValue_ULInt);
   IF "EingangM19P2" THEN "DB_Station19_Port2".TagAtHead := TRUE; END_IF;
   IF NOT "EingangM19P2" THEN "DB_Station19_Port2".TagAtHead := FALSE; END_IF;
   "DB_Station19_Port2".CurrentValue := S_CONV(IN := "DB_Station19_Port2".CurrentValue_ULInt);
END_REGION

REGION Network 27: Station20/Port1
   // Setzen der Werte für den entsprechenden Datenbaustein
   CALC(in1 := "ByteM20P1.1",
        in2 := "ByteM20P1.2",
        in3 := "ByteM20P1.3",
        in4 := "ByteM20P1.4",
        in5 := "ByteM20P1.5",
        in6 := "ByteM20P1.6",
        in7 := "ByteM20P1.7",
        in8 := "ByteM20P1.8",
        in9 := 256,
        out => "DB_Station20_Port1".CurrentValue_ULInt);
   IF "EingangM20P1" THEN "DB_Station20_Port1".TagAtHead := TRUE; END_IF;
   IF NOT "EingangM20P1" THEN "DB_Station20_Port1".TagAtHead := FALSE; END_IF;
   "DB_Station20_Port1".CurrentValue := S_CONV(IN := "DB_Station20_Port1".CurrentValue_ULInt);
END_REGION

REGION Network 28: Parametrierung des IO-Devices (nicht verwendet) - geht analog für den Master
   // CAP ist bei Balluff immer 255
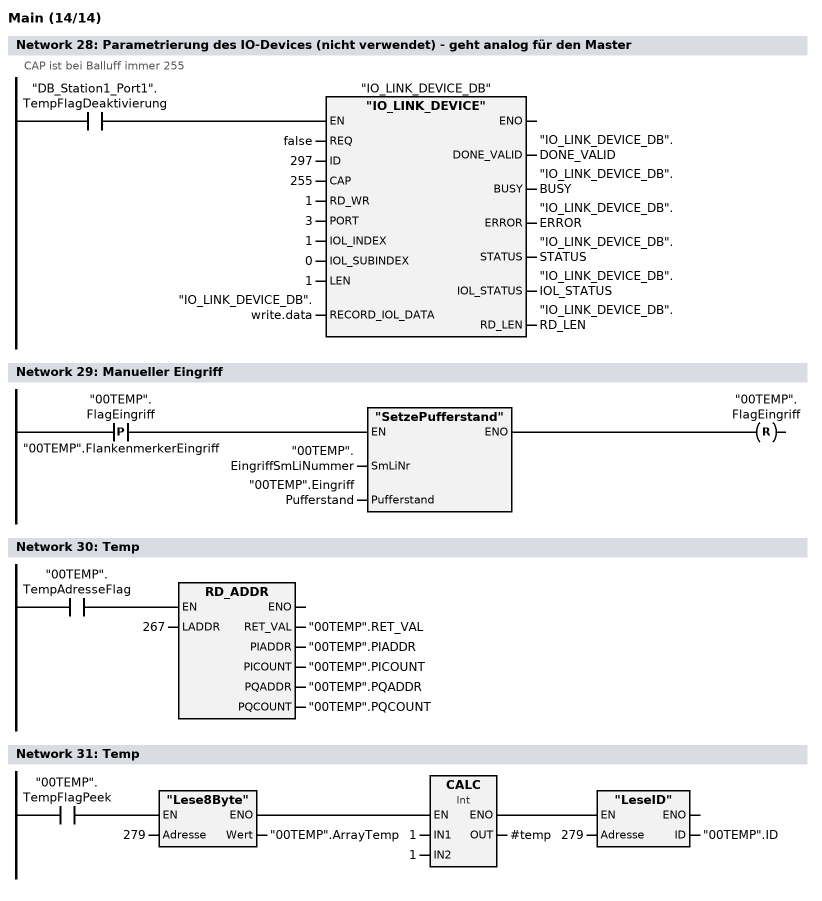
   RUNG wire#powerrail
      Contact( "DB_Station1_Port1".TempFlagDeaktivierung )
      "IO_LINK_DEVICE_DB"(REQ := false, ID := 297, CAP := 255, RD_WR := 1, PORT := 3, IOL_INDEX := 1, IOL_SUBINDEX := 0, LEN := 1, RECORD_IOL_DATA := "IO_LINK_DEVICE_DB".write.data, DONE_VALID => "IO_LINK_DEVICE_DB".DONE_VALID, BUSY => "IO_LINK_DEVICE_DB".BUSY, ERROR => "IO_LINK_DEVICE_DB".ERROR, STATUS => "IO_LINK_DEVICE_DB".STATUS, IOL_STATUS => "IO_LINK_DEVICE_DB".IOL_STATUS, RD_LEN => "IO_LINK_DEVICE_DB".RD_LEN)
   END_RUNG
   // the same network as SCL:
   IF "DB_Station1_Port1".TempFlagDeaktivierung THEN
       "IO_LINK_DEVICE_DB"(REQ := false,   // "IO_LINK_DEVICE"
                           ID := 297,
                           CAP := 255,
                           RD_WR := 1,
                           PORT := 3,
                           IOL_INDEX := 1,
                           IOL_SUBINDEX := 0,
                           LEN := 1,
                           RECORD_IOL_DATA := "IO_LINK_DEVICE_DB".write.data,
                           DONE_VALID => "IO_LINK_DEVICE_DB".DONE_VALID,
                           BUSY => "IO_LINK_DEVICE_DB".BUSY,
                           ERROR => "IO_LINK_DEVICE_DB".ERROR,
                           STATUS => "IO_LINK_DEVICE_DB".STATUS,
                           IOL_STATUS => "IO_LINK_DEVICE_DB".IOL_STATUS,
                           RD_LEN => "IO_LINK_DEVICE_DB".RD_LEN);
   END_IF;
END_REGION

REGION Network 29: Manueller Eingriff
   RUNG wire#powerrail
      P_Contact(operand := "00TEMP".FlagEingriff, bit := "00TEMP".FlankenmerkerEingriff)
      "SetzePufferstand"(SmLiNr := "00TEMP".EingriffSmLiNummer, Pufferstand := "00TEMP".EingriffPufferstand)
      R_Coil( "00TEMP".FlagEingriff )
   END_RUNG
   // the same network as SCL:
   #_w1 := "00TEMP".FlagEingriff AND NOT "00TEMP".FlankenmerkerEingriff;   // rising edge of "00TEMP".FlagEingriff
   "00TEMP".FlankenmerkerEingriff := "00TEMP".FlagEingriff;
   "SetzePufferstand"(EN := #_w1,
                      SmLiNr := "00TEMP".EingriffSmLiNummer,
                      Pufferstand := "00TEMP".EingriffPufferstand,
                      ENO => #_w2);
   IF #_w2 THEN "00TEMP".FlagEingriff := FALSE; END_IF;
END_REGION

REGION Network 30: Temp
   IF "00TEMP".TempAdresseFlag THEN
       "00TEMP".RET_VAL := RD_ADDR(LADDR := 267,
                               PIADDR => "00TEMP".PIADDR,
                               PICount => "00TEMP".PICOUNT,
                               PQADDR => "00TEMP".PQADDR,
                               PQCount => "00TEMP".PQCOUNT);
   END_IF;
END_REGION

REGION Network 31: Temp
   "Lese8Byte"(EN := "00TEMP".TempFlagPeek, Adresse := 279, Wert => "00TEMP".ArrayTemp, ENO => #_w1);
   IF #_w1 THEN
       CALC(in1 := 1, in2 := 1, out => #temp);
       "LeseID"(Adresse := 279, ID => "00TEMP".ID);
   END_IF;
END_REGION

REGION Network 32 (SCL): Temp zum Aktivieren
   IF "Test".FlagAk THEN
       "Test".Req := true;
       "Test".RetValD_ACT_DP2 := D_ACT_DP(LADDR := "Station7~IODevice", MODE := 1, REQ := "Test".Req, BUSY => "Test".Busy2);
       "Test".FlagAk := false;
   END_IF;
END_REGION
END_ORGANIZATION_BLOCK

ORGANIZATION_BLOCK "Status"   // OB55, LAD, Status
TITLE = "DP:status_alarm"
{ S7_Optimized_Access := 'TRUE' }
VERSION : 0.1
   VAR_INPUT
      LADDR : Hw_Io;   // Hardware identifier
      Slot : UInt;   // Slot number
      Specifier : Word;   // alarm specifier out of the alarm telegram
   END_VAR
BEGIN

REGION Network 1
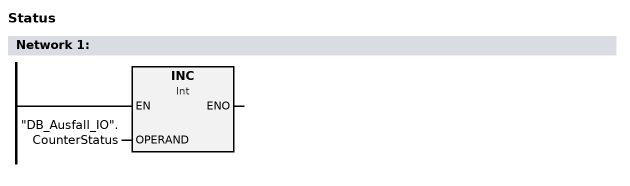
   RUNG wire#powerrail
      { S7_Templates := "DestType := Int" } Inc( "DB_Ausfall_IO".CounterStatus )
   END_RUNG
   // the same network as SCL:
   "DB_Ausfall_IO".CounterStatus := "DB_Ausfall_IO".CounterStatus + 1;
END_REGION
END_ORGANIZATION_BLOCK

ORGANIZATION_BLOCK "Profile"   // OB57, LAD, Profile
TITLE = "DP:manufacture_alarm"
{ S7_Optimized_Access := 'TRUE' }
VERSION : 0.1
   VAR_INPUT
      LADDR : Hw_Io;   // Hardware identifier
      Slot : UInt;   // Slot number
      Specifier : Word;   // alarm specifier out of the alarm telegram
   END_VAR
BEGIN

REGION Network 1
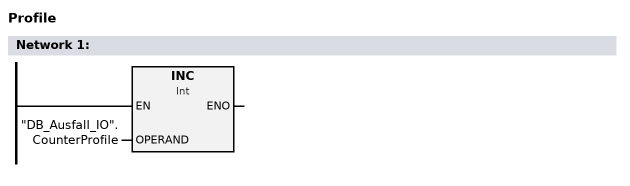
   RUNG wire#powerrail
      { S7_Templates := "DestType := Int" } Inc( "DB_Ausfall_IO".CounterProfile )
   END_RUNG
   // the same network as SCL:
   "DB_Ausfall_IO".CounterProfile := "DB_Ausfall_IO".CounterProfile + 1;
END_REGION
END_ORGANIZATION_BLOCK

ORGANIZATION_BLOCK "Time error interrupt"   // OB80, LAD, TimeErrorInterrupt
{ S7_Optimized_Access := 'TRUE' }
VERSION : 0.1
   VAR_INPUT
      Fault_ID : Byte;   // Fault identifier
      Csg_OBnr : OB_Any;   // Number of OB causing the error
      Csg_Prio : UInt;   // Priority of OB causing the error
   END_VAR
BEGIN
END_ORGANIZATION_BLOCK

ORGANIZATION_BLOCK "Pull or plug of modules"   // OB83, LAD, PullPlug
{ S7_Optimized_Access := 'TRUE' }
VERSION : 0.1
   VAR_INPUT
      LADDR : Hw_Io;   // Hardware identifier
      Event_Class : Byte;   // 16#38/39: module inserted, removed
      Fault_ID : Byte;   // Fault identifier
   END_VAR
BEGIN

REGION Network 1
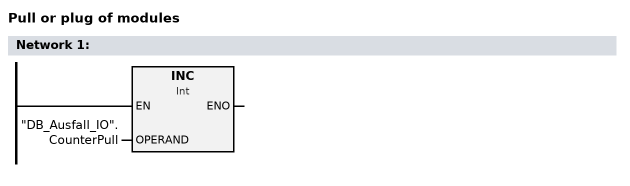
   RUNG wire#powerrail
      { S7_Templates := "DestType := Int" } Inc( "DB_Ausfall_IO".CounterPull )
   END_RUNG
   // the same network as SCL:
   "DB_Ausfall_IO".CounterPull := "DB_Ausfall_IO".CounterPull + 1;
END_REGION
END_ORGANIZATION_BLOCK

ORGANIZATION_BLOCK "Rack or station failure"   // OB86, LAD, RackStationFailure
{ S7_Optimized_Access := 'TRUE' }
VERSION : 0.1
   VAR_INPUT
      LADDR : Hw_Device;   // Hardware identifier
      Event_Class : Byte;   // Event class
      Fault_ID : Byte;   // Fault identifier
   END_VAR
   VAR_TEMP
      Auftrag : Byte;
      Start : Bool;
      Busy : Bool;
      RET_Val : Int;
   END_VAR
   VAR_TEMP   // added for the SCL form of the ladder/FBD networks
      _w1 : Bool;
      _w2 : Bool;
      _w3 : Bool;
      _w4 : Bool;
      _w5 : Bool;
   END_VAR
BEGIN

REGION Network 1
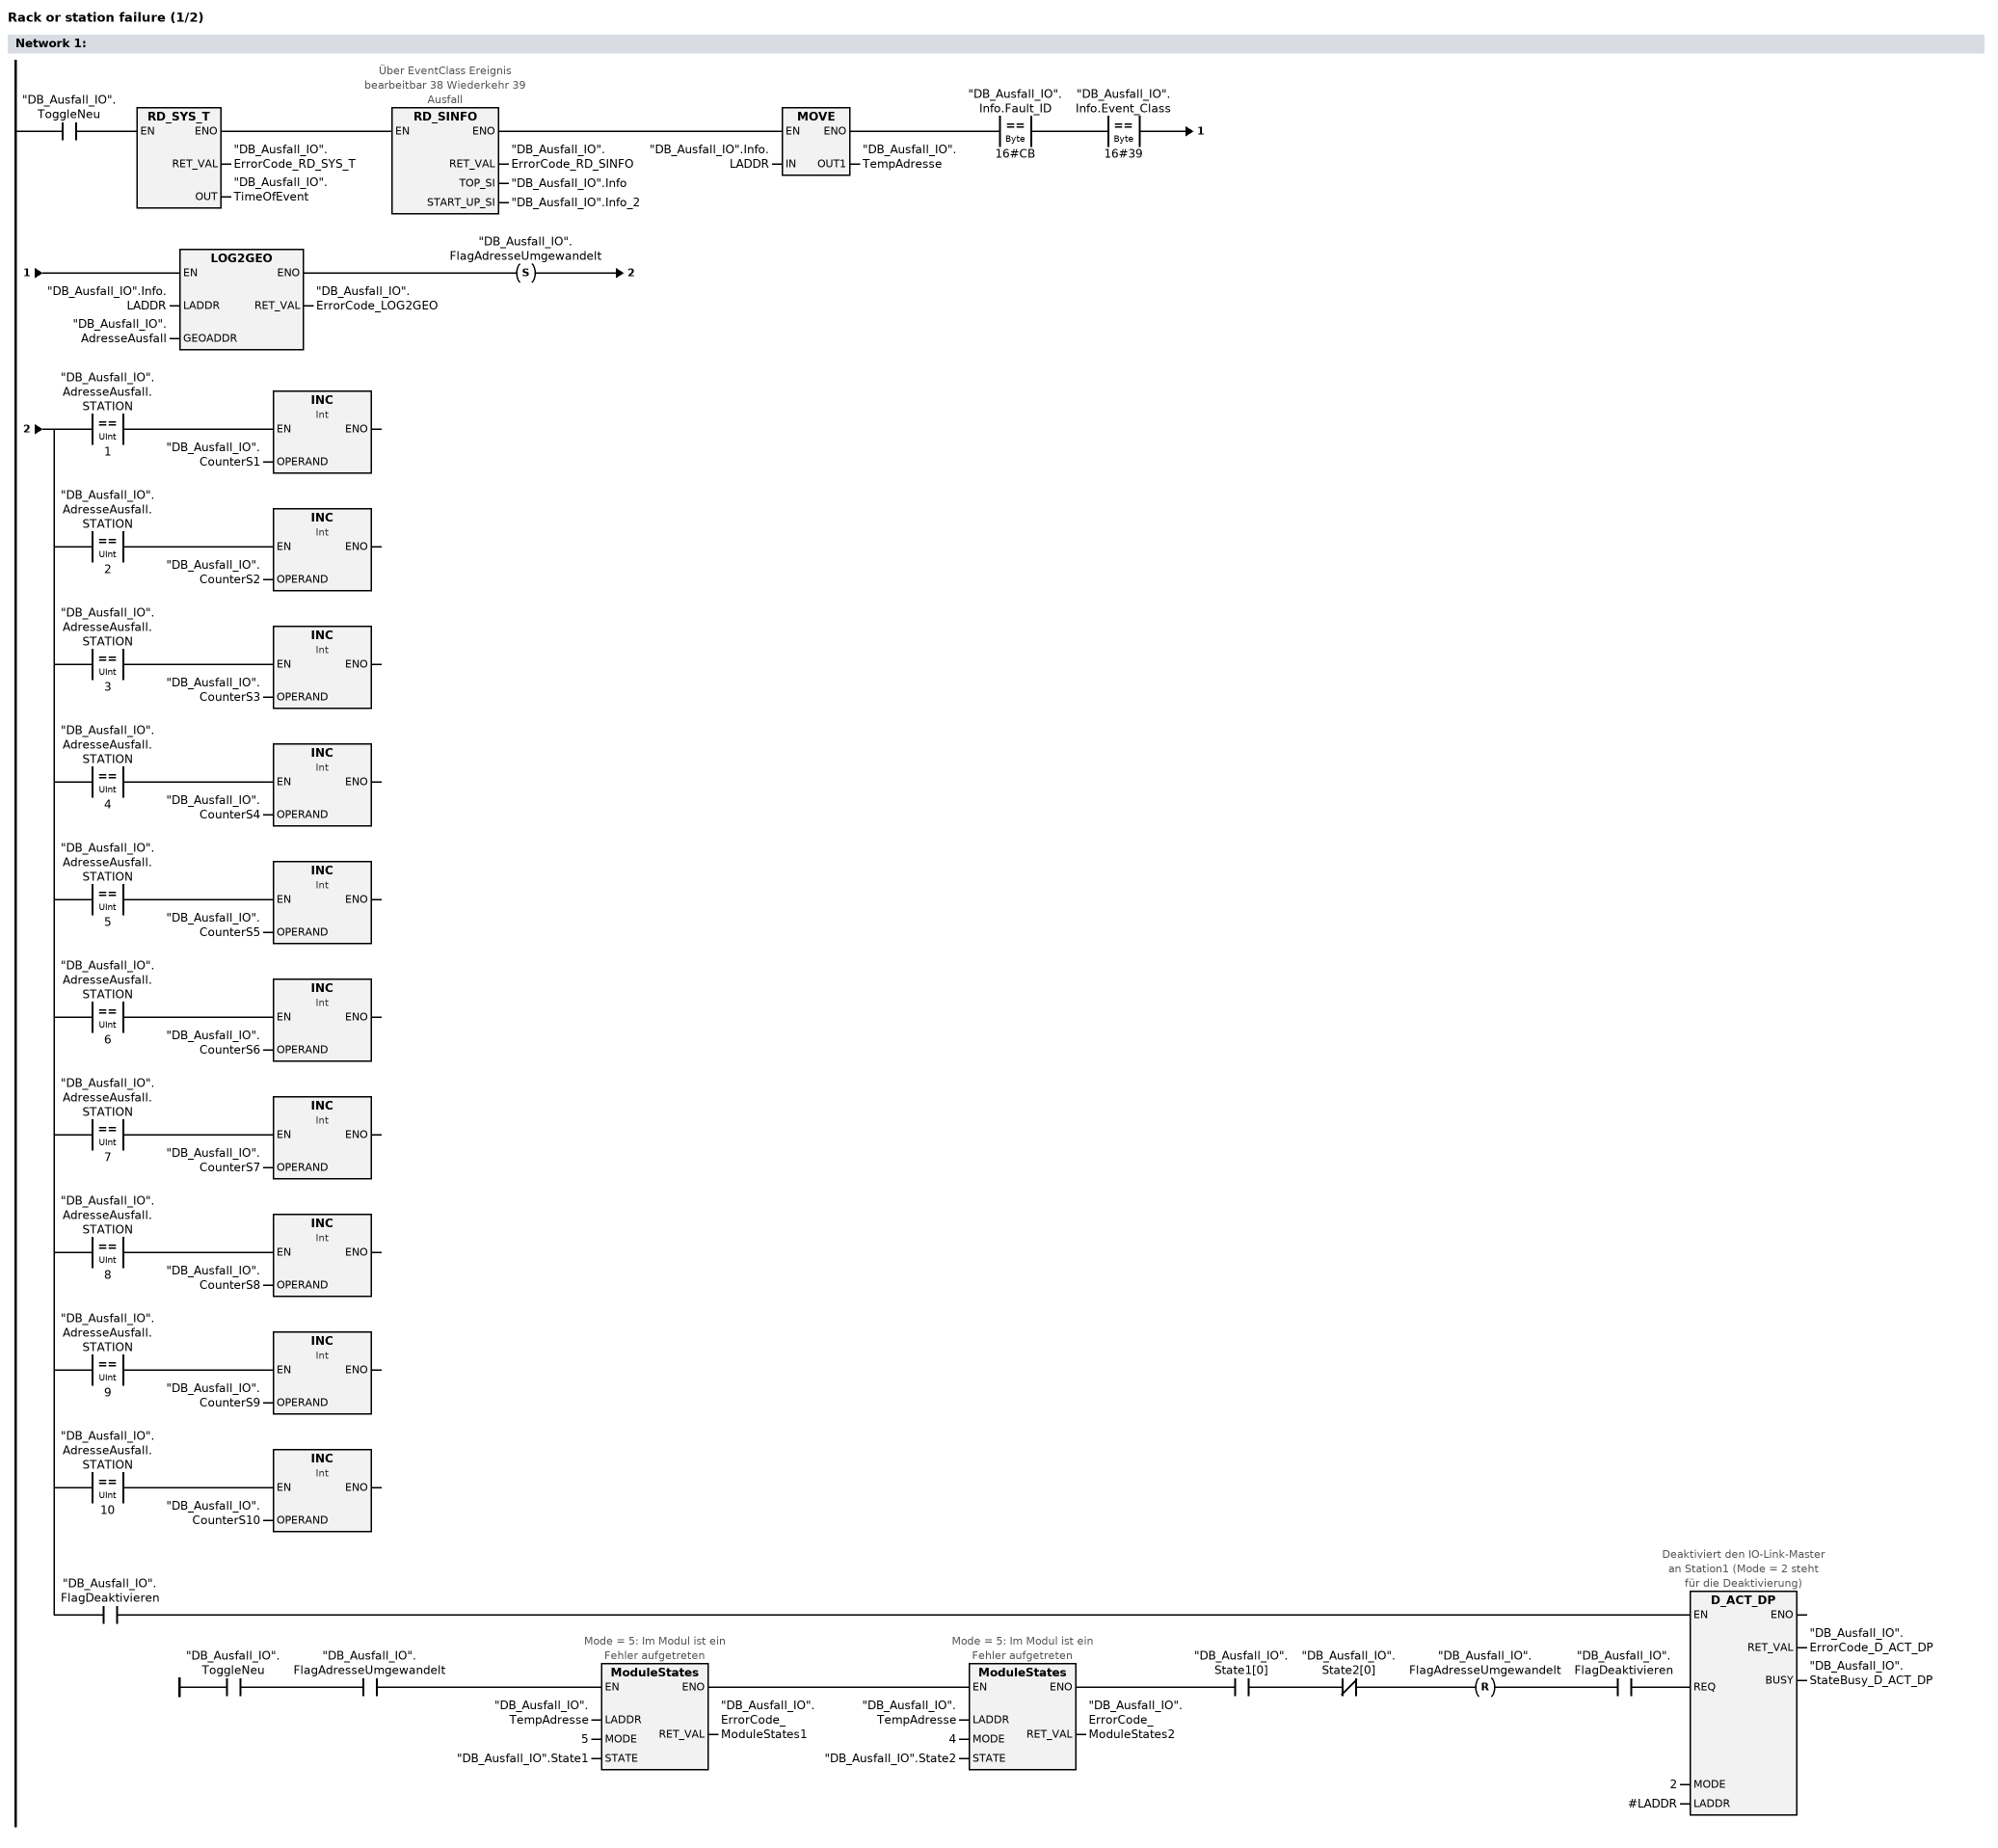
   // no SCL statement known for ModuleStates: written as a call
   // ENO of a box is taken as its EN; it also drops when the box reports an error
   #_w1 := "DB_Ausfall_IO".ToggleNeu;
   IF #_w1 THEN
       "DB_Ausfall_IO".ErrorCode_RD_SYS_T := RD_SYS_T(OUT => "DB_Ausfall_IO".TimeOfEvent);
       "DB_Ausfall_IO".ErrorCode_RD_SINFO := RD_SINFO(TOP_SI => "DB_Ausfall_IO".Info,   // Über EventClass Ereignis bearbeitbar 38 Wiederkehr 39 Ausfall
                               START_UP_SI => "DB_Ausfall_IO".Info_2);
       "DB_Ausfall_IO".TempAdresse := "DB_Ausfall_IO".Info.LADDR;
   END_IF;
   #_w2 := #_w1 AND ("DB_Ausfall_IO".Info.Fault_ID = 16#CB) AND ("DB_Ausfall_IO".Info.Event_Class = 16#39);
   IF #_w2 THEN
       "DB_Ausfall_IO".ErrorCode_LOG2GEO := LOG2GEO(LADDR := "DB_Ausfall_IO".Info.LADDR,
                               GEOADDR := "DB_Ausfall_IO".AdresseAusfall);
       "DB_Ausfall_IO".FlagAdresseUmgewandelt := TRUE;
   END_IF;
   IF #_w2 AND ("DB_Ausfall_IO".AdresseAusfall.STATION = 1) THEN
       "DB_Ausfall_IO".CounterS1 := "DB_Ausfall_IO".CounterS1 + 1;
   END_IF;
   IF #_w2 AND ("DB_Ausfall_IO".AdresseAusfall.STATION = 2) THEN
       "DB_Ausfall_IO".CounterS2 := "DB_Ausfall_IO".CounterS2 + 1;
   END_IF;
   IF #_w2 AND ("DB_Ausfall_IO".AdresseAusfall.STATION = 3) THEN
       "DB_Ausfall_IO".CounterS3 := "DB_Ausfall_IO".CounterS3 + 1;
   END_IF;
   IF #_w2 AND ("DB_Ausfall_IO".AdresseAusfall.STATION = 4) THEN
       "DB_Ausfall_IO".CounterS4 := "DB_Ausfall_IO".CounterS4 + 1;
   END_IF;
   IF #_w2 AND ("DB_Ausfall_IO".AdresseAusfall.STATION = 5) THEN
       "DB_Ausfall_IO".CounterS5 := "DB_Ausfall_IO".CounterS5 + 1;
   END_IF;
   IF #_w2 AND ("DB_Ausfall_IO".AdresseAusfall.STATION = 6) THEN
       "DB_Ausfall_IO".CounterS6 := "DB_Ausfall_IO".CounterS6 + 1;
   END_IF;
   IF #_w2 AND ("DB_Ausfall_IO".AdresseAusfall.STATION = 7) THEN
       "DB_Ausfall_IO".CounterS7 := "DB_Ausfall_IO".CounterS7 + 1;
   END_IF;
   IF #_w2 AND ("DB_Ausfall_IO".AdresseAusfall.STATION = 8) THEN
       "DB_Ausfall_IO".CounterS8 := "DB_Ausfall_IO".CounterS8 + 1;
   END_IF;
   IF #_w2 AND ("DB_Ausfall_IO".AdresseAusfall.STATION = 9) THEN
       "DB_Ausfall_IO".CounterS9 := "DB_Ausfall_IO".CounterS9 + 1;
   END_IF;
   IF #_w2 AND ("DB_Ausfall_IO".AdresseAusfall.STATION = 10) THEN
       "DB_Ausfall_IO".CounterS10 := "DB_Ausfall_IO".CounterS10 + 1;
   END_IF;
   #_w3 := "DB_Ausfall_IO".ToggleNeu AND "DB_Ausfall_IO".FlagAdresseUmgewandelt;
   #_w4 := #_w2 AND "DB_Ausfall_IO".FlagDeaktivieren;
   IF #_w3 THEN
       "DB_Ausfall_IO".ErrorCode_ModuleStates1 := ModuleStates(LADDR := "DB_Ausfall_IO".TempAdresse,   // Mode = 5: Im Modul ist ein Fehler aufgetreten
                               MODE := 5,
                               STATE := "DB_Ausfall_IO".State1);
       "DB_Ausfall_IO".ErrorCode_ModuleStates2 := ModuleStates(LADDR := "DB_Ausfall_IO".TempAdresse,   // Mode = 5: Im Modul ist ein Fehler aufgetreten
                               MODE := 4,
                               STATE := "DB_Ausfall_IO".State2);
   END_IF;
   #_w5 := #_w3 AND "DB_Ausfall_IO".State1[0] AND NOT "DB_Ausfall_IO".State2[0];
   IF #_w5 THEN "DB_Ausfall_IO".FlagAdresseUmgewandelt := FALSE; END_IF;
   IF #_w4 THEN
       "DB_Ausfall_IO".ErrorCode_D_ACT_DP := D_ACT_DP(REQ := #_w5 AND "DB_Ausfall_IO".FlagDeaktivieren,   // Deaktiviert den IO-Link-Master an Station1 (Mode = 2 steht für die Deaktivierung)
                               MODE := 2,
                               LADDR := #LADDR,
                               BUSY => "DB_Ausfall_IO".StateBusy_D_ACT_DP);
   END_IF;
END_REGION

REGION Network 2
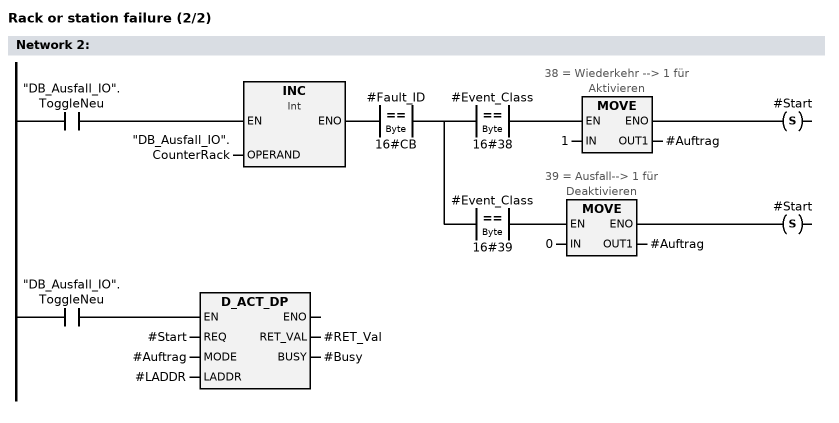
   IF "DB_Ausfall_IO".ToggleNeu THEN "DB_Ausfall_IO".CounterRack := "DB_Ausfall_IO".CounterRack + 1; END_IF;
   #_w1 := "DB_Ausfall_IO".ToggleNeu AND (#Fault_ID = 16#CB);
   IF #_w1 AND (#Event_Class = 16#38) THEN
       #Auftrag := 1;   // 38 = Wiederkehr --> 1 für Aktivieren
       #Start := TRUE;
   END_IF;
   IF #_w1 AND (#Event_Class = 16#39) THEN
       #Auftrag := 0;   // 39 = Ausfall--> 1 für Deaktivieren
       #Start := TRUE;
   END_IF;
   IF "DB_Ausfall_IO".ToggleNeu THEN
       #RET_Val := D_ACT_DP(REQ := #Start, MODE := #Auftrag, LADDR := #LADDR, BUSY => #Busy);
   END_IF;
END_REGION
END_ORGANIZATION_BLOCK

ORGANIZATION_BLOCK "Startup"   // OB100, LAD, Startup
TITLE = "Complete Restart"
{ S7_Optimized_Access := 'TRUE' }
VERSION : 0.1
// Beim Hochfahren der SPS auszuführen
   VAR_INPUT
      LostRetentive : Bool;   // True if retentive data are lost
      LostRTC : Bool;   // True if date and time are lost
   END_VAR
   VAR_TEMP
      i : Int;
      Adresse : Hw_Device;
      KennungDeaktivieren : USInt;
      KennungVorhanden : UInt;
      KennungFehler : UInt;
      ZustandVorhanden : Bool;
      ZustandFehler : Bool;
      temp : Int;
      BoolReq : Bool;
      busy : Bool;
   END_VAR
BEGIN

REGION Network 1: Startwerte der Puffer setzen
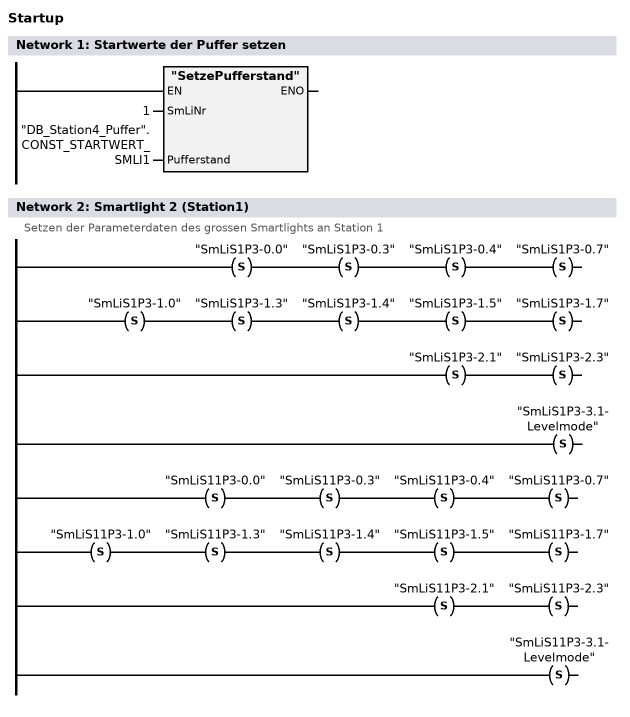
   RUNG wire#powerrail
      "SetzePufferstand"(SmLiNr := 1, Pufferstand := "DB_Station4_Puffer".CONST_STARTWERT_SMLI1)
   END_RUNG
   // the same network as SCL:
   "SetzePufferstand"(SmLiNr := 1, Pufferstand := "DB_Station4_Puffer".CONST_STARTWERT_SMLI1);
END_REGION

REGION Network 2: Smartlight 2 (Station1)
   // Setzen der Parameterdaten des grossen Smartlights an Station 1
   RUNG wire#powerrail
      S_Coil( "SmLiS1P3-0.0" )
      S_Coil( "SmLiS1P3-0.3" )
      S_Coil( "SmLiS1P3-0.4" )
      S_Coil( "SmLiS1P3-0.7" )
   END_RUNG
   RUNG wire#powerrail
      S_Coil( "SmLiS1P3-1.0" )
      S_Coil( "SmLiS1P3-1.3" )
      S_Coil( "SmLiS1P3-1.4" )
      S_Coil( "SmLiS1P3-1.5" )
      S_Coil( "SmLiS1P3-1.7" )
   END_RUNG
   RUNG wire#powerrail
      S_Coil( "SmLiS1P3-2.1" )
      S_Coil( "SmLiS1P3-2.3" )
   END_RUNG
   RUNG wire#powerrail
      S_Coil( "SmLiS1P3-3.1-Levelmode" )
   END_RUNG
   RUNG wire#powerrail
      S_Coil( "SmLiS11P3-0.0" )
      S_Coil( "SmLiS11P3-0.3" )
      S_Coil( "SmLiS11P3-0.4" )
      S_Coil( "SmLiS11P3-0.7" )
   END_RUNG
   RUNG wire#powerrail
      S_Coil( "SmLiS11P3-1.0" )
      S_Coil( "SmLiS11P3-1.3" )
      S_Coil( "SmLiS11P3-1.4" )
      S_Coil( "SmLiS11P3-1.5" )
      S_Coil( "SmLiS11P3-1.7" )
   END_RUNG
   RUNG wire#powerrail
      S_Coil( "SmLiS11P3-2.1" )
      S_Coil( "SmLiS11P3-2.3" )
   END_RUNG
   RUNG wire#powerrail
      S_Coil( "SmLiS11P3-3.1-Levelmode" )
   END_RUNG
   // the same network as SCL:
   "SmLiS1P3-0.0" := TRUE;
   "SmLiS1P3-0.3" := TRUE;
   "SmLiS1P3-0.4" := TRUE;
   "SmLiS1P3-0.7" := TRUE;
   "SmLiS1P3-1.0" := TRUE;
   "SmLiS1P3-1.3" := TRUE;
   "SmLiS1P3-1.4" := TRUE;
   "SmLiS1P3-1.5" := TRUE;
   "SmLiS1P3-1.7" := TRUE;
   "SmLiS1P3-2.1" := TRUE;
   "SmLiS1P3-2.3" := TRUE;
   "SmLiS1P3-3.1-Levelmode" := TRUE;
   "SmLiS11P3-0.0" := TRUE;
   "SmLiS11P3-0.3" := TRUE;
   "SmLiS11P3-0.4" := TRUE;
   "SmLiS11P3-0.7" := TRUE;
   "SmLiS11P3-1.0" := TRUE;
   "SmLiS11P3-1.3" := TRUE;
   "SmLiS11P3-1.4" := TRUE;
   "SmLiS11P3-1.5" := TRUE;
   "SmLiS11P3-1.7" := TRUE;
   "SmLiS11P3-2.1" := TRUE;
   "SmLiS11P3-2.3" := TRUE;
   "SmLiS11P3-3.1-Levelmode" := TRUE;
END_REGION

REGION Network 3 (SCL): Granularitaet der Smartlights an Station 1 setzen
   FOR #i  := 1 TO 2 DO
       "BestimmeGranularitaet"(#i);
   END_FOR;
END_REGION

REGION Network 4 (SCL): Speicherung der HW-Adressen der IO-Link Master
   "DB_Konstanten".HW_Adressen[0] := "Station1~IODevice";
   "DB_Konstanten".HW_Adressen[1] := "Station2~IODevice";
   "DB_Konstanten".HW_Adressen[2] := "Station3~IODevice";
   "DB_Konstanten".HW_Adressen[3] := "Station4~IODevice";
   "DB_Konstanten".HW_Adressen[4] := "Station5~IODevice";
   "DB_Konstanten".HW_Adressen[5] := "Station6~IODevice";
   "DB_Konstanten".HW_Adressen[6] := "Station7~IODevice";
   "DB_Konstanten".HW_Adressen[7] := "Station8~IODevice";
   "DB_Konstanten".HW_Adressen[8] := "Station9~IODevice";
   "DB_Konstanten".HW_Adressen[9] := "Station10~IODevice";
   "DB_Konstanten".HW_Adressen[10] := "Station11~IODevice";
   "DB_Konstanten".HW_Adressen[11] := "Station12~IODevice";
   "DB_Konstanten".HW_Adressen[12] := "Station13~IODevice";
   "DB_Konstanten".HW_Adressen[13] := "Station15~IODevice";
   "DB_Konstanten".HW_Adressen[14] := "Station16~IODevice";
   "DB_Konstanten".HW_Adressen[15] := "Station17~IODevice";
   "DB_Konstanten".HW_Adressen[16] := "Station19~IODevice";
   "DB_Konstanten".HW_Adressen[17] := "Station20~IODevice";
   "DB_Konstanten".HW_Adressen[18] := "BVS-SC~IODevice";
END_REGION

REGION Network 5 (SCL): Deaktivierung nicht erreichbarer IO-Link Master
   #KennungDeaktivieren := 2;
   #KennungVorhanden := 4;
   #KennungFehler := 5;
   FOR #i := 0 TO "DB_Konstanten"."Anzahl Adressen" - 1 DO
       #Adresse := "DB_Konstanten".HW_Adressen[#i];
       IF #Adresse = 0 THEN
           CONTINUE;
       END_IF;
       #temp := ModuleStates(LADDR := #Adresse,MODE := #KennungVorhanden,STATE := #ZustandVorhanden);
       #temp := ModuleStates(LADDR := #Adresse, MODE := #KennungFehler, STATE := #ZustandFehler);
       IF (NOT #ZustandVorhanden) AND (#ZustandFehler) THEN
           #BoolReq := true;
           #temp := D_ACT_DP(REQ := #BoolReq, LADDR := #Adresse, MODE := #KennungDeaktivieren, BUSY =>#busy);
           #BoolReq := false;
           WHILE #busy = true DO
               #temp := D_ACT_DP(REQ := #BoolReq, LADDR := #Adresse, MODE := #KennungDeaktivieren, BUSY => #busy);
           END_WHILE;
           RE_TRIGR();
      END_IF;
   END_FOR;
END_REGION
END_ORGANIZATION_BLOCK

ORGANIZATION_BLOCK "IO access error"   // OB122, LAD, IOAccessError
{ S7_Optimized_Access := 'TRUE' }
VERSION : 0.1
   VAR_INPUT
      BlockNr : UInt;   // Number of causing block
      Reaction : USInt;   // 0:ignore, 1:substitute, 2:skip
      Fault_ID : Byte;   // 16#42:reading, 16#43:writing
      BlockType : USInt;   // 16#01:OB, 16#02:FC, 16#03:FB, 16#04:SFC, 16#05:SFB, 16#06:DB: Type of block causing the error
      Area : USInt;   // 16#81:I, 16#82:Q: IO area where the IOaccess error occured
      DBNr : DB_ANY;   // Reserved for system
      Csg_OBNr : OB_Any;   // Number of OB causing the error
      Csg_Prio : USInt;   // Priority of OB causing the error
      Width : USInt;   // 0:bit, 1:byte, 2:word, 3:dword, 4:lword
   END_VAR
BEGIN

REGION Network 1
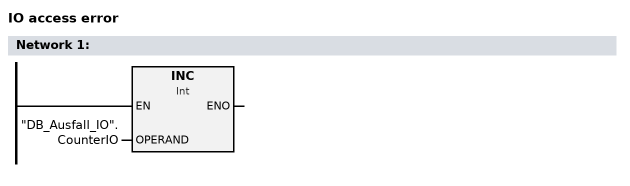
   RUNG wire#powerrail
      { S7_Templates := "DestType := Int" } Inc( "DB_Ausfall_IO".CounterIO )
   END_RUNG
   // the same network as SCL:
   "DB_Ausfall_IO".CounterIO := "DB_Ausfall_IO".CounterIO + 1;
END_REGION
END_ORGANIZATION_BLOCK